END_WHILE
enumerator.Dispose();
END_METHOD

PROPERTY PUBLIC Address : PVOID
GET
Address := ADR(activeData);
END_GET
END_PROPERTY

PROPERTY PUBLIC BaseDatatype : I_Datatype
GET
BaseDatatype := baseType;
END_GET
END_PROPERTY

METHOD PUBLIC ClearReference
VAR_INPUT
END_VAR
activeData REF= localData;
SetElementReference();
END_METHOD

PROPERTY PUBLIC Size : UDINT
GET
Size := SIZEOF(activeData);
END_GET
END_PROPERTY

METHOD PUBLIC TryGetElementAsDatatypeByIndex : BOOL
VAR_INPUT
	Index : DINT;
	Destination : REFERENCE TO I_Datatype;
END_VAR
IF Index < lbound OR Index > ubound THEN
	RETURN;
END_IF

Destination := elements[Index];
TryGetElementAsDatatypeByIndex := TRUE;
END_METHOD

METHOD PUBLIC TryGetLowerBound : BOOL
VAR_INPUT
	Dimention : UDINT;
	Destination : REFERENCE TO DINT;
END_VAR
IF Dimention = 1 THEN
	Destination := lBound;
	TryGetLowerBound := TRUE;
END_IF
END_METHOD

METHOD PUBLIC TryGetUpperBound : BOOL
VAR_INPUT
	Dimention : UDINT;
	Destination : REFERENCE TO DINT;
END_VAR
IF Dimention = 1 THEN
	Destination := uBound;
	TryGetUpperBound := TRUE;
END_IF
END_METHOD

METHOD PUBLIC Clone : I_Datatype
VAR
    pClone : POINTER TO _Array0to3OfINT;
END_VAR
pClone := __NEW(_Array0to3OfINT());
pClone^.Value := Value;
Clone := pClone^;
END_METHOD

METHOD PUBLIC MakeReferenceTo
VAR_INPUT
	ReferenceTarget : REFERENCE TO ARRAY [lBound..uBound] OF INT;
END_VAR
activeData REF= ReferenceTarget;
SetElementReference();
END_METHOD

METHOD TryMakeReferenceTo : BOOL
VAR_INPUT
	Target : I_Datatype;
END_VAR
VAR
	targetAsArray : I_ArrayDatatype;
	pTargetData : POINTER TO ARRAY [lBound..uBound] OF INT;
END_VAR
IF NOT Target.TryResolveAsArrayDatatype(targetAsArray) THEN
	RETURN;
END_IF

IF NOT (targetAsArray.Identifier = Identifier) THEN
	RETURN;
END_IF

pTargetData := Target.Address;
activeData REF= pTargetData^;
SetElementReference();
TryMakeReferenceTo := TRUE;
END_METHOD

PROPERTY PUBLIC Value : REFERENCE TO ARRAY [lBound..uBound] OF INT;
GET
Value ref= activeData;
END_GET
END_PROPERTY

END_FUNCTION_BLOCK

// Datatypes/Aliases/_TcVnVector4_LREAL
{attribute 'linkalways'} 
{attribute 'no_explicit_call' := 'This FB is a CLASS and must be accessed using methods or properties'}
{attribute 'enable_dynamic_creation'}
FUNCTION_BLOCK _TcVnVector4_LREAL EXTENDS AliasDatatypeBase
VAR
	localData : TcVnVector4_LREAL;
	activeData : REFERENCE TO TcVnVector4_LREAL REF= localData;
	aliasBaseDatatype : _Array0to3OfLREAL;
END_VAR

METHOD PROTECTED SetBaseDatatypeReference
VAR_INPUT
END_VAR
aliasBaseDatatype.MakeReferenceTo(activeData);
END_METHOD

PROPERTY PUBLIC Address : PVOID
GET
Address := ADR(activeData);
END_GET
END_PROPERTY

METHOD PUBLIC ClearReference
VAR_INPUT
END_VAR
activeData REF= localData;
SetBaseDatatypeReference();
END_METHOD

PROPERTY PUBLIC Size : UDINT
GET
Size := SIZEOF(activeData);
END_GET
END_PROPERTY

METHOD FB_init : BOOL
VAR_INPUT
	bInitRetains : BOOL; // if TRUE, the retain variables are initialized (warm start / cold start)
	bInCopyCode : BOOL;  // if TRUE, the instance afterwards gets moved into the copy code (online change)
	//InitialValue : <type>; // if possible, not all values can be initialized
END_VAR
//localData := InitialValue; // if possible, not all values can be initialized
SetBaseDatatypeReference();
AddBaseDatatype(aliasBaseDatatype);
END_METHOD

METHOD PUBLIC Clone : I_Datatype
VAR
    pClone : POINTER TO _TcVnVector4_LREAL;
END_VAR
pClone := __NEW(_TcVnVector4_LREAL);
Clone := pClone^;
END_METHOD

PROPERTY PUBLIC Identifier : T_MAXSTRING
GET
Identifier := 'TcVnVector4_LREAL';
END_GET
END_PROPERTY

METHOD PUBLIC MakeReferenceTo
VAR_INPUT
	ReferenceTarget : REFERENCE TO TcVnVector4_LREAL;
END_VAR
activeData REF= ReferenceTarget;
SetBaseDatatypeReference();
END_METHOD

METHOD TryMakeReferenceTo : BOOL
VAR_INPUT
	Target : I_Datatype;
END_VAR
VAR
	targetAsAlias : I_AliasDatatype;
	pTargetData : POINTER TO TcVnVector4_LREAL;
END_VAR
IF NOT Target.TryResolveAsAliasDatatype(targetAsAlias) THEN
	RETURN;
END_IF

IF targetAsAlias.Identifier <> Identifier THEN
	RETURN;
END_IF

pTargetData := Target.Address;
activeData REF= pTargetData^;
SetBaseDatatypeReference();
TryMakeReferenceTo := TRUE;
END_METHOD

PROPERTY PUBLIC Value : REFERENCE TO TcVnVector4_LREAL
GET
Value REF= activeData;
END_GET
END_PROPERTY

END_FUNCTION_BLOCK

// Datatypes/Aliases/_TcVnVector4_SINT
{attribute 'linkalways'} 
{attribute 'no_explicit_call' := 'This FB is a CLASS and must be accessed using methods or properties'}
{attribute 'enable_dynamic_creation'}
FUNCTION_BLOCK _TcVnVector4_SINT EXTENDS AliasDatatypeBase
VAR
	localData : TcVnVector4_SINT;
	activeData : REFERENCE TO TcVnVector4_SINT REF= localData;
	aliasBaseDatatype : _Array0to3OfSINT;
END_VAR

METHOD PROTECTED SetBaseDatatypeReference
VAR_INPUT
END_VAR
aliasBaseDatatype.MakeReferenceTo(activeData);
END_METHOD

PROPERTY PUBLIC Address : PVOID
GET
Address := ADR(activeData);
END_GET
END_PROPERTY

METHOD PUBLIC ClearReference
VAR_INPUT
END_VAR
activeData REF= localData;
SetBaseDatatypeReference();
END_METHOD

PROPERTY PUBLIC Size : UDINT
GET
Size := SIZEOF(activeData);
END_GET
END_PROPERTY

METHOD FB_init : BOOL
VAR_INPUT
	bInitRetains : BOOL; // if TRUE, the retain variables are initialized (warm start / cold start)
	bInCopyCode : BOOL;  // if TRUE, the instance afterwards gets moved into the copy code (online change)
	//InitialValue : <type>; // if possible, not all values can be initialized
END_VAR
//localData := InitialValue; // if possible, not all values can be initialized
SetBaseDatatypeReference();
AddBaseDatatype(aliasBaseDatatype);
END_METHOD

METHOD PUBLIC Clone : I_Datatype
VAR
    pClone : POINTER TO _TcVnVector4_SINT;
END_VAR
pClone := __NEW(_TcVnVector4_SINT);
Clone := pClone^;
END_METHOD

PROPERTY PUBLIC Identifier : T_MAXSTRING
GET
Identifier := 'TcVnVector4_SINT';
END_GET
END_PROPERTY

METHOD PUBLIC MakeReferenceTo
VAR_INPUT
	ReferenceTarget : REFERENCE TO TcVnVector4_SINT;
END_VAR
activeData REF= ReferenceTarget;
SetBaseDatatypeReference();
END_METHOD

METHOD TryMakeReferenceTo : BOOL
VAR_INPUT
	Target : I_Datatype;
END_VAR
VAR
	targetAsAlias : I_AliasDatatype;
	pTargetData : POINTER TO TcVnVector4_SINT;
END_VAR
IF NOT Target.TryResolveAsAliasDatatype(targetAsAlias) THEN
	RETURN;
END_IF

IF targetAsAlias.Identifier <> Identifier THEN
	RETURN;
END_IF

pTargetData := Target.Address;
activeData REF= pTargetData^;
SetBaseDatatypeReference();
TryMakeReferenceTo := TRUE;
END_METHOD

PROPERTY PUBLIC Value : REFERENCE TO TcVnVector4_SINT
GET
Value REF= activeData;
END_GET
END_PROPERTY

END_FUNCTION_BLOCK

// Datatypes/Arrays/_Array0to3OfSINT
{attribute 'linkalways'} 
{attribute 'no_explicit_call' := 'This FB is a CLASS and must be accessed using methods or properties'}
{attribute 'enable_dynamic_creation'}
FUNCTION_BLOCK _Array0to3OfSINT EXTENDS ArrayDatatypeBase_1D
VAR CONSTANT
	lBound : DINT := 0;
	uBound : DINT := 3;
END_VAR
VAR
	localData : ARRAY [lBound..uBound] OF SINT;
	activeData : REFERENCE TO ARRAY [lBound..uBound] OF SINT REF= localData;
	elements : ARRAY [lBound..uBound] OF _SINT(0);
	baseType : _SINT(0);
END_VAR

METHOD FB_init : BOOL
VAR_INPUT
	bInitRetains : BOOL; // if TRUE, the retain variables are initialized (warm start / cold start)
	bInCopyCode : BOOL;  // if TRUE, the instance afterwards gets moved into the copy code (online change)
END_VAR
SetElementReference();
END_METHOD

METHOD PROTECTED OnSerializeArrayValues
VAR_INPUT
	Serializer : I_Serializer;
END_VAR
VAR
	i : DINT;
END_VAR
FOR i := lBound TO uBound DO
	elements[i].SerializeWith(Serializer);
END_FOR
END_METHOD

METHOD PROTECTED SetElementReference
VAR_INPUT
END_VAR
VAR
	i : DINT;
END_VAR
FOR i := lBound TO uBound DO
	elements[i].MakeReferenceTo(activeData[i]);
END_FOR
END_METHOD

METHOD PROTECTED TryDeserializeArrayValues : BOOL
VAR_INPUT
	Deserializer : I_Deserializer;
	Feedback : I_DeserializerFeedback;
END_VAR
VAR
	enumerator : I_DeserializerArrayForwardEnumerator;
	i : DINT;
END_VAR
enumerator := Deserializer.GetArrayEnumerator();
i := lBound;

WHILE enumerator.MoveNext() AND i <= uBound DO
	
	IF NOT elements[i].TryDeserializeFrom(enumerator.Current, Feedback) THEN
		EXIT;
	END_IF
	i := i + 1;

END_WHILE
enumerator.Dispose();
END_METHOD

PROPERTY PUBLIC Address : PVOID
GET
Address := ADR(activeData);
END_GET
END_PROPERTY

PROPERTY PUBLIC BaseDatatype : I_Datatype
GET
BaseDatatype := baseType;
END_GET
END_PROPERTY

METHOD PUBLIC ClearReference
VAR_INPUT
END_VAR
activeData REF= localData;
SetElementReference();
END_METHOD

PROPERTY PUBLIC Size : UDINT
GET
Size := SIZEOF(activeData);
END_GET
END_PROPERTY

METHOD PUBLIC TryGetElementAsDatatypeByIndex : BOOL
VAR_INPUT
	Index : DINT;
	Destination : REFERENCE TO I_Datatype;
END_VAR
IF Index < lbound OR Index > ubound THEN
	RETURN;
END_IF

Destination := elements[Index];
TryGetElementAsDatatypeByIndex := TRUE;
END_METHOD

METHOD PUBLIC TryGetLowerBound : BOOL
VAR_INPUT
	Dimention : UDINT;
	Destination : REFERENCE TO DINT;
END_VAR
IF Dimention = 1 THEN
	Destination := lBound;
	TryGetLowerBound := TRUE;
END_IF
END_METHOD

METHOD PUBLIC TryGetUpperBound : BOOL
VAR_INPUT
	Dimention : UDINT;
	Destination : REFERENCE TO DINT;
END_VAR
IF Dimention = 1 THEN
	Destination := uBound;
	TryGetUpperBound := TRUE;
END_IF
END_METHOD

METHOD PUBLIC Clone : I_Datatype
VAR
    pClone : POINTER TO _Array0to3OfSINT;
END_VAR
pClone := __NEW(_Array0to3OfSINT());
pClone^.Value := Value;
Clone := pClone^;
END_METHOD

METHOD PUBLIC MakeReferenceTo
VAR_INPUT
	ReferenceTarget : REFERENCE TO ARRAY [lBound..uBound] OF SINT;
END_VAR
activeData REF= ReferenceTarget;
SetElementReference();
END_METHOD

METHOD TryMakeReferenceTo : BOOL
VAR_INPUT
	Target : I_Datatype;
END_VAR
VAR
	targetAsArray : I_ArrayDatatype;
	pTargetData : POINTER TO ARRAY [lBound..uBound] OF SINT;
END_VAR
IF NOT Target.TryResolveAsArrayDatatype(targetAsArray) THEN
	RETURN;
END_IF

IF NOT (targetAsArray.Identifier = Identifier) THEN
	RETURN;
END_IF

pTargetData := Target.Address;
activeData REF= pTargetData^;
SetElementReference();
TryMakeReferenceTo := TRUE;
END_METHOD

PROPERTY PUBLIC Value : REFERENCE TO ARRAY [lBound..uBound] OF SINT;
GET
Value ref= activeData;
END_GET
END_PROPERTY

END_FUNCTION_BLOCK

// Datatypes/Aliases/_TcVnVector4_UINT
{attribute 'linkalways'} 
{attribute 'no_explicit_call' := 'This FB is a CLASS and must be accessed using methods or properties'}
{attribute 'enable_dynamic_creation'}
FUNCTION_BLOCK _TcVnVector4_UINT EXTENDS AliasDatatypeBase
VAR
	localData : TcVnVector4_UINT;
	activeData : REFERENCE TO TcVnVector4_UINT REF= localData;
	aliasBaseDatatype : _Array0to3OfUINT;
END_VAR

METHOD PROTECTED SetBaseDatatypeReference
VAR_INPUT
END_VAR
aliasBaseDatatype.MakeReferenceTo(activeData);
END_METHOD

PROPERTY PUBLIC Address : PVOID
GET
Address := ADR(activeData);
END_GET
END_PROPERTY

METHOD PUBLIC ClearReference
VAR_INPUT
END_VAR
activeData REF= localData;
SetBaseDatatypeReference();
END_METHOD

PROPERTY PUBLIC Size : UDINT
GET
Size := SIZEOF(activeData);
END_GET
END_PROPERTY

METHOD FB_init : BOOL
VAR_INPUT
	bInitRetains : BOOL; // if TRUE, the retain variables are initialized (warm start / cold start)
	bInCopyCode : BOOL;  // if TRUE, the instance afterwards gets moved into the copy code (online change)
	//InitialValue : <type>; // if possible, not all values can be initialized
END_VAR
//localData := InitialValue; // if possible, not all values can be initialized
SetBaseDatatypeReference();
AddBaseDatatype(aliasBaseDatatype);
END_METHOD

METHOD PUBLIC Clone : I_Datatype
VAR
    pClone : POINTER TO _TcVnVector4_UINT;
END_VAR
pClone := __NEW(_TcVnVector4_UINT);
Clone := pClone^;
END_METHOD

PROPERTY PUBLIC Identifier : T_MAXSTRING
GET
Identifier := 'TcVnVector4_UINT';
END_GET
END_PROPERTY

METHOD PUBLIC MakeReferenceTo
VAR_INPUT
	ReferenceTarget : REFERENCE TO TcVnVector4_UINT;
END_VAR
activeData REF= ReferenceTarget;
SetBaseDatatypeReference();
END_METHOD

METHOD TryMakeReferenceTo : BOOL
VAR_INPUT
	Target : I_Datatype;
END_VAR
VAR
	targetAsAlias : I_AliasDatatype;
	pTargetData : POINTER TO TcVnVector4_UINT;
END_VAR
IF NOT Target.TryResolveAsAliasDatatype(targetAsAlias) THEN
	RETURN;
END_IF

IF targetAsAlias.Identifier <> Identifier THEN
	RETURN;
END_IF

pTargetData := Target.Address;
activeData REF= pTargetData^;
SetBaseDatatypeReference();
TryMakeReferenceTo := TRUE;
END_METHOD

PROPERTY PUBLIC Value : REFERENCE TO TcVnVector4_UINT
GET
Value REF= activeData;
END_GET
END_PROPERTY

END_FUNCTION_BLOCK

// Datatypes/Arrays/_Array0to3OfUINT
{attribute 'linkalways'} 
{attribute 'no_explicit_call' := 'This FB is a CLASS and must be accessed using methods or properties'}
{attribute 'enable_dynamic_creation'}
FUNCTION_BLOCK _Array0to3OfUINT EXTENDS ArrayDatatypeBase_1D
VAR CONSTANT
	lBound : DINT := 0;
	uBound : DINT := 3;
END_VAR
VAR
	localData : ARRAY [lBound..uBound] OF UINT;
	activeData : REFERENCE TO ARRAY [lBound..uBound] OF UINT REF= localData;
	elements : ARRAY [lBound..uBound] OF _UINT(0);
	baseType : _UINT(0);
END_VAR

METHOD FB_init : BOOL
VAR_INPUT
	bInitRetains : BOOL; // if TRUE, the retain variables are initialized (warm start / cold start)
	bInCopyCode : BOOL;  // if TRUE, the instance afterwards gets moved into the copy code (online change)
END_VAR
SetElementReference();
END_METHOD

METHOD PROTECTED OnSerializeArrayValues
VAR_INPUT
	Serializer : I_Serializer;
END_VAR
VAR
	i : DINT;
END_VAR
FOR i := lBound TO uBound DO
	elements[i].SerializeWith(Serializer);
END_FOR
END_METHOD

METHOD PROTECTED SetElementReference
VAR_INPUT
END_VAR
VAR
	i : DINT;
END_VAR
FOR i := lBound TO uBound DO
	elements[i].MakeReferenceTo(activeData[i]);
END_FOR
END_METHOD

METHOD PROTECTED TryDeserializeArrayValues : BOOL
VAR_INPUT
	Deserializer : I_Deserializer;
	Feedback : I_DeserializerFeedback;
END_VAR
VAR
	enumerator : I_DeserializerArrayForwardEnumerator;
	i : DINT;
END_VAR
enumerator := Deserializer.GetArrayEnumerator();
i := lBound;

WHILE enumerator.MoveNext() AND i <= uBound DO
	
	IF NOT elements[i].TryDeserializeFrom(enumerator.Current, Feedback) THEN
		EXIT;
	END_IF
	i := i + 1;

END_WHILE
enumerator.Dispose();
END_METHOD

PROPERTY PUBLIC Address : PVOID
GET
Address := ADR(activeData);
END_GET
END_PROPERTY

PROPERTY PUBLIC BaseDatatype : I_Datatype
GET
BaseDatatype := baseType;
END_GET
END_PROPERTY

METHOD PUBLIC ClearReference
VAR_INPUT
END_VAR
activeData REF= localData;
SetElementReference();
END_METHOD

PROPERTY PUBLIC Size : UDINT
GET
Size := SIZEOF(activeData);
END_GET
END_PROPERTY

METHOD PUBLIC TryGetElementAsDatatypeByIndex : BOOL
VAR_INPUT
	Index : DINT;
	Destination : REFERENCE TO I_Datatype;
END_VAR
IF Index < lbound OR Index > ubound THEN
	RETURN;
END_IF

Destination := elements[Index];
TryGetElementAsDatatypeByIndex := TRUE;
END_METHOD

METHOD PUBLIC TryGetLowerBound : BOOL
VAR_INPUT
	Dimention : UDINT;
	Destination : REFERENCE TO DINT;
END_VAR
IF Dimention = 1 THEN
	Destination := lBound;
	TryGetLowerBound := TRUE;
END_IF
END_METHOD

METHOD PUBLIC TryGetUpperBound : BOOL
VAR_INPUT
	Dimention : UDINT;
	Destination : REFERENCE TO DINT;
END_VAR
IF Dimention = 1 THEN
	Destination := uBound;
	TryGetUpperBound := TRUE;
END_IF
END_METHOD

METHOD PUBLIC Clone : I_Datatype
VAR
    pClone : POINTER TO _Array0to3OfUINT;
END_VAR
pClone := __NEW(_Array0to3OfUINT());
pClone^.Value := Value;
Clone := pClone^;
END_METHOD

METHOD PUBLIC MakeReferenceTo
VAR_INPUT
	ReferenceTarget : REFERENCE TO ARRAY [lBound..uBound] OF UINT;
END_VAR
activeData REF= ReferenceTarget;
SetElementReference();
END_METHOD

METHOD TryMakeReferenceTo : BOOL
VAR_INPUT
	Target : I_Datatype;
END_VAR
VAR
	targetAsArray : I_ArrayDatatype;
	pTargetData : POINTER TO ARRAY [lBound..uBound] OF UINT;
END_VAR
IF NOT Target.TryResolveAsArrayDatatype(targetAsArray) THEN
	RETURN;
END_IF

IF NOT (targetAsArray.Identifier = Identifier) THEN
	RETURN;
END_IF

pTargetData := Target.Address;
activeData REF= pTargetData^;
SetElementReference();
TryMakeReferenceTo := TRUE;
END_METHOD

PROPERTY PUBLIC Value : REFERENCE TO ARRAY [lBound..uBound] OF UINT;
GET
Value ref= activeData;
END_GET
END_PROPERTY

END_FUNCTION_BLOCK

// Datatypes/Aliases/_TcVnVector4_USINT
{attribute 'linkalways'} 
{attribute 'no_explicit_call' := 'This FB is a CLASS and must be accessed using methods or properties'}
{attribute 'enable_dynamic_creation'}
FUNCTION_BLOCK _TcVnVector4_USINT EXTENDS AliasDatatypeBase
VAR
	localData : TcVnVector4_USINT;
	activeData : REFERENCE TO TcVnVector4_USINT REF= localData;
	aliasBaseDatatype : _Array0to3OfUSINT;
END_VAR

METHOD PROTECTED SetBaseDatatypeReference
VAR_INPUT
END_VAR
aliasBaseDatatype.MakeReferenceTo(activeData);
END_METHOD

PROPERTY PUBLIC Address : PVOID
GET
Address := ADR(activeData);
END_GET
END_PROPERTY

METHOD PUBLIC ClearReference
VAR_INPUT
END_VAR
activeData REF= localData;
SetBaseDatatypeReference();
END_METHOD

PROPERTY PUBLIC Size : UDINT
GET
Size := SIZEOF(activeData);
END_GET
END_PROPERTY

METHOD FB_init : BOOL
VAR_INPUT
	bInitRetains : BOOL; // if TRUE, the retain variables are initialized (warm start / cold start)
	bInCopyCode : BOOL;  // if TRUE, the instance afterwards gets moved into the copy code (online change)
	//InitialValue : <type>; // if possible, not all values can be initialized
END_VAR
//localData := InitialValue; // if possible, not all values can be initialized
SetBaseDatatypeReference();
AddBaseDatatype(aliasBaseDatatype);
END_METHOD

METHOD PUBLIC Clone : I_Datatype
VAR
    pClone : POINTER TO _TcVnVector4_USINT;
END_VAR
pClone := __NEW(_TcVnVector4_USINT);
Clone := pClone^;
END_METHOD

PROPERTY PUBLIC Identifier : T_MAXSTRING
GET
Identifier := 'TcVnVector4_USINT';
END_GET
END_PROPERTY

METHOD PUBLIC MakeReferenceTo
VAR_INPUT
	ReferenceTarget : REFERENCE TO TcVnVector4_USINT;
END_VAR
activeData REF= ReferenceTarget;
SetBaseDatatypeReference();
END_METHOD

METHOD TryMakeReferenceTo : BOOL
VAR_INPUT
	Target : I_Datatype;
END_VAR
VAR
	targetAsAlias : I_AliasDatatype;
	pTargetData : POINTER TO TcVnVector4_USINT;
END_VAR
IF NOT Target.TryResolveAsAliasDatatype(targetAsAlias) THEN
	RETURN;
END_IF

IF targetAsAlias.Identifier <> Identifier THEN
	RETURN;
END_IF

pTargetData := Target.Address;
activeData REF= pTargetData^;
SetBaseDatatypeReference();
TryMakeReferenceTo := TRUE;
END_METHOD

PROPERTY PUBLIC Value : REFERENCE TO TcVnVector4_USINT
GET
Value REF= activeData;
END_GET
END_PROPERTY

END_FUNCTION_BLOCK

// Datatypes/Arrays/_Array0to3OfUSINT
{attribute 'linkalways'} 
{attribute 'no_explicit_call' := 'This FB is a CLASS and must be accessed using methods or properties'}
{attribute 'enable_dynamic_creation'}
FUNCTION_BLOCK _Array0to3OfUSINT EXTENDS ArrayDatatypeBase_1D
VAR CONSTANT
	lBound : DINT := 0;
	uBound : DINT := 3;
END_VAR
VAR
	localData : ARRAY [lBound..uBound] OF USINT;
	activeData : REFERENCE TO ARRAY [lBound..uBound] OF USINT REF= localData;
	elements : ARRAY [lBound..uBound] OF _USINT(0);
	baseType : _USINT(0);
END_VAR

METHOD FB_init : BOOL
VAR_INPUT
	bInitRetains : BOOL; // if TRUE, the retain variables are initialized (warm start / cold start)
	bInCopyCode : BOOL;  // if TRUE, the instance afterwards gets moved into the copy code (online change)
END_VAR
SetElementReference();
END_METHOD

METHOD PROTECTED OnSerializeArrayValues
VAR_INPUT
	Serializer : I_Serializer;
END_VAR
VAR
	i : DINT;
END_VAR
FOR i := lBound TO uBound DO
	elements[i].SerializeWith(Serializer);
END_FOR
END_METHOD

METHOD PROTECTED SetElementReference
VAR_INPUT
END_VAR
VAR
	i : DINT;
END_VAR
FOR i := lBound TO uBound DO
	elements[i].MakeReferenceTo(activeData[i]);
END_FOR
END_METHOD

METHOD PROTECTED TryDeserializeArrayValues : BOOL
VAR_INPUT
	Deserializer : I_Deserializer;
	Feedback : I_DeserializerFeedback;
END_VAR
VAR
	enumerator : I_DeserializerArrayForwardEnumerator;
	i : DINT;
END_VAR
enumerator := Deserializer.GetArrayEnumerator();
i := lBound;

WHILE enumerator.MoveNext() AND i <= uBound DO
	
	IF NOT elements[i].TryDeserializeFrom(enumerator.Current, Feedback) THEN
		EXIT;
	END_IF
	i := i + 1;

END_WHILE
enumerator.Dispose();
END_METHOD

PROPERTY PUBLIC Address : PVOID
GET
Address := ADR(activeData);
END_GET
END_PROPERTY

PROPERTY PUBLIC BaseDatatype : I_Datatype
GET
BaseDatatype := baseType;
END_GET
END_PROPERTY

METHOD PUBLIC ClearReference
VAR_INPUT
END_VAR
activeData REF= localData;
SetElementReference();
END_METHOD

PROPERTY PUBLIC Size : UDINT
GET
Size := SIZEOF(activeData);
END_GET
END_PROPERTY

METHOD PUBLIC TryGetElementAsDatatypeByIndex : BOOL
VAR_INPUT
	Index : DINT;
	Destination : REFERENCE TO I_Datatype;
END_VAR
IF Index < lbound OR Index > ubound THEN
	RETURN;
END_IF

Destination := elements[Index];
TryGetElementAsDatatypeByIndex := TRUE;
END_METHOD

METHOD PUBLIC TryGetLowerBound : BOOL
VAR_INPUT
	Dimention : UDINT;
	Destination : REFERENCE TO DINT;
END_VAR
IF Dimention = 1 THEN
	Destination := lBound;
	TryGetLowerBound := TRUE;
END_IF
END_METHOD

METHOD PUBLIC TryGetUpperBound : BOOL
VAR_INPUT
	Dimention : UDINT;
	Destination : REFERENCE TO DINT;
END_VAR
IF Dimention = 1 THEN
	Destination := uBound;
	TryGetUpperBound := TRUE;
END_IF
END_METHOD

METHOD PUBLIC Clone : I_Datatype
VAR
    pClone : POINTER TO _Array0to3OfUSINT;
END_VAR
pClone := __NEW(_Array0to3OfUSINT());
pClone^.Value := Value;
Clone := pClone^;
END_METHOD

METHOD PUBLIC MakeReferenceTo
VAR_INPUT
	ReferenceTarget : REFERENCE TO ARRAY [lBound..uBound] OF USINT;
END_VAR
activeData REF= ReferenceTarget;
SetElementReference();
END_METHOD

METHOD TryMakeReferenceTo : BOOL
VAR_INPUT
	Target : I_Datatype;
END_VAR
VAR
	targetAsArray : I_ArrayDatatype;
	pTargetData : POINTER TO ARRAY [lBound..uBound] OF USINT;
END_VAR
IF NOT Target.TryResolveAsArrayDatatype(targetAsArray) THEN
	RETURN;
END_IF

IF NOT (targetAsArray.Identifier = Identifier) THEN
	RETURN;
END_IF

pTargetData := Target.Address;
activeData REF= pTargetData^;
SetElementReference();
TryMakeReferenceTo := TRUE;
END_METHOD

PROPERTY PUBLIC Value : REFERENCE TO ARRAY [lBound..uBound] OF USINT;
GET
Value ref= activeData;
END_GET
END_PROPERTY

END_FUNCTION_BLOCK

// Datatypes/Arrays/_Array0to1_0to2OfLREAL
{attribute 'linkalways'} 
{attribute 'no_explicit_call' := 'This FB is a CLASS and must be accessed using methods or properties'}
{attribute 'enable_dynamic_creation'}
FUNCTION_BLOCK _Array0to1_0to2OfLREAL EXTENDS ArrayDatatypeBase_2D
VAR CONSTANT
	lBoundD1 : DINT := 0;
	uBoundD1 : DINT := 1;
	lBoundD2 : DINT := 0;
	uBoundD2 : DINT := 2;
END_VAR
VAR
	localData : ARRAY [lBoundD1..uBoundD1,lBoundD2..uBoundD2] OF LREAL;
	activeData : REFERENCE TO ARRAY [lBoundD1..uBoundD1,lBoundD2..uBoundD2] OF LREAL REF= localData;
	elements : ARRAY [lBoundD1..uBoundD1,lBoundD2..uBoundD2] OF _LREAL(0);
	baseType : _LREAL(0);
END_VAR

METHOD FB_init : BOOL
VAR_INPUT
	bInitRetains : BOOL; // if TRUE, the retain variables are initialized (warm start / cold start)
	bInCopyCode : BOOL;  // if TRUE, the instance afterwards gets moved into the copy code (online change)
END_VAR
SetElementReference();
END_METHOD

METHOD PROTECTED OnSerializeArrayValues
VAR_INPUT
	Serializer : I_Serializer;
END_VAR
VAR
	i, j : DINT;
END_VAR
FOR i := lBoundD1 TO uBoundD1 DO
	Serializer.StartArray();
	FOR j := lBoundD2 TO uBoundD2 DO
		elements[i, j].SerializeWith(Serializer);
	END_FOR
	Serializer.EndArray();
END_FOR
END_METHOD

METHOD PROTECTED SetElementReference
VAR_INPUT
END_VAR
VAR
	i, j : DINT;
END_VAR
FOR i := lBoundD1 TO uBoundD1 DO
	FOR j := lBoundD2 TO uBoundD2 DO
		elements[i, j].MakeReferenceTo(activeData[i, j]);
	END_FOR
END_FOR
END_METHOD

METHOD PROTECTED TryDeserializeArrayValues : BOOL
VAR_INPUT
	Deserializer : I_Deserializer;
	Feedback : I_DeserializerFeedback;
END_VAR
VAR
	enumeratorD1 : I_DeserializerArrayForwardEnumerator;
	enumeratorD2 : I_DeserializerArrayForwardEnumerator;
	i, j : DINT;
END_VAR
enumeratorD1 := Deserializer.GetArrayEnumerator();
i := lBoundD1;

WHILE enumeratorD1.MoveNext() AND i <= uBoundD1 DO
	
	enumeratorD2 := enumeratorD1.Current.GetArrayEnumerator();
	j := lBoundD2;
	
	WHILE enumeratorD2.MoveNext() AND j <= uBoundD2 DO
	
		IF NOT elements[i, j].TryDeserializeFrom(enumeratorD2.Current, Feedback) THEN
			EXIT;
		END_IF
		
		j := j + 1;
	
	END_WHILE
	enumeratorD2.Dispose();

	i := i + 1;

END_WHILE
enumeratorD1.Dispose();
END_METHOD

PROPERTY PUBLIC Address : PVOID
GET
Address := ADR(activeData);
END_GET
END_PROPERTY

PROPERTY PUBLIC BaseDatatype : I_Datatype
GET
BaseDatatype := baseType;
END_GET
END_PROPERTY

METHOD PUBLIC ClearReference
VAR_INPUT
END_VAR
activeData REF= localData;
SetElementReference();
END_METHOD

PROPERTY PUBLIC Size : UDINT
GET
Size := SIZEOF(activeData);
END_GET
END_PROPERTY

METHOD PUBLIC TryGetElementAsDatatypeByIndex : BOOL
VAR_INPUT
	Index1 : DINT;
	Index2 : DINT;
	Destination : REFERENCE TO I_Datatype;
END_VAR
IF Index1 < lboundD1 OR Index1 > uboundD1 THEN
	RETURN;
END_IF

IF Index2 < lboundD2 OR Index2 > uboundD2 THEN
	RETURN;
END_IF

Destination := elements[Index1, Index2];
TryGetElementAsDatatypeByIndex := TRUE;
END_METHOD

METHOD PUBLIC TryGetLowerBound : BOOL
VAR_INPUT
	Dimention : UDINT;
	Destination : REFERENCE TO DINT;
END_VAR
CASE Dimention OF
	
	1:	Destination := lBoundD1;
		TryGetLowerBound := TRUE;
		RETURN;
	
	2:	Destination := lBoundD2;
		TryGetLowerBound := TRUE;
		RETURN;

END_CASE
END_METHOD

METHOD PUBLIC TryGetUpperBound : BOOL
VAR_INPUT
	Dimention : UDINT;
	Destination : REFERENCE TO DINT;
END_VAR
CASE Dimention OF
	
	1:	Destination := uBoundD1;
		TryGetUpperBound := TRUE;
		RETURN;
	
	2:	Destination := uBoundD2;
		TryGetUpperBound := TRUE;
		RETURN;

END_CASE
END_METHOD

METHOD PUBLIC Clone : I_Datatype
VAR
    pClone : POINTER TO _Array0to1_0to2OfLREAL;
END_VAR
pClone := __NEW(_Array0to1_0to2OfLREAL());
pClone^.Value := Value;
Clone := pClone^;
END_METHOD

METHOD PUBLIC MakeReferenceTo
VAR_INPUT
	ReferenceTarget : REFERENCE TO ARRAY [lBoundD1..uBoundD1,lBoundD2..uBoundD2] OF LREAL;
END_VAR
activeData REF= ReferenceTarget;
SetElementReference();
END_METHOD

METHOD TryMakeReferenceTo : BOOL
VAR_INPUT
	Target : I_Datatype;
END_VAR
VAR
	targetAsArray : I_ArrayDatatype;
	pTargetData : POINTER TO ARRAY [lBoundD1..uBoundD1,lBoundD2..uBoundD2] OF LREAL;
END_VAR
IF NOT Target.TryResolveAsArrayDatatype(targetAsArray) THEN
	RETURN;
END_IF

IF NOT (targetAsArray.Identifier = Identifier) THEN
	RETURN;
END_IF

pTargetData := Target.Address;
activeData REF= pTargetData^;
SetElementReference();
TryMakeReferenceTo := TRUE;
END_METHOD

PROPERTY PUBLIC Value : REFERENCE TO ARRAY [lBoundD1..uBoundD1,lBoundD2..uBoundD2] OF LREAL;
GET
Value ref= activeData;
END_GET
END_PROPERTY

END_FUNCTION_BLOCK

// Datatypes/Arrays/_Array0to2_0to2OfLREAL
{attribute 'linkalways'} 
{attribute 'no_explicit_call' := 'This FB is a CLASS and must be accessed using methods or properties'}
{attribute 'enable_dynamic_creation'}
FUNCTION_BLOCK _Array0to2_0to2OfLREAL EXTENDS ArrayDatatypeBase_2D
VAR CONSTANT
	lBoundD1 : DINT := 0;
	uBoundD1 : DINT := 2;
	lBoundD2 : DINT := 0;
	uBoundD2 : DINT := 2;
END_VAR
VAR
	localData : ARRAY [lBoundD1..uBoundD1,lBoundD2..uBoundD2] OF LREAL;
	activeData : REFERENCE TO ARRAY [lBoundD1..uBoundD1,lBoundD2..uBoundD2] OF LREAL REF= localData;
	elements : ARRAY [lBoundD1..uBoundD1,lBoundD2..uBoundD2] OF _LREAL(0);
	baseType : _LREAL(0);
END_VAR

METHOD FB_init : BOOL
VAR_INPUT
	bInitRetains : BOOL; // if TRUE, the retain variables are initialized (warm start / cold start)
	bInCopyCode : BOOL;  // if TRUE, the instance afterwards gets moved into the copy code (online change)
END_VAR
SetElementReference();
END_METHOD

METHOD PROTECTED OnSerializeArrayValues
VAR_INPUT
	Serializer : I_Serializer;
END_VAR
VAR
	i, j : DINT;
END_VAR
FOR i := lBoundD1 TO uBoundD1 DO
	Serializer.StartArray();
	FOR j := lBoundD2 TO uBoundD2 DO
		elements[i, j].SerializeWith(Serializer);
	END_FOR
	Serializer.EndArray();
END_FOR
END_METHOD

METHOD PROTECTED SetElementReference
VAR_INPUT
END_VAR
VAR
	i, j : DINT;
END_VAR
FOR i := lBoundD1 TO uBoundD1 DO
	FOR j := lBoundD2 TO uBoundD2 DO
		elements[i, j].MakeReferenceTo(activeData[i, j]);
	END_FOR
END_FOR
END_METHOD

METHOD PROTECTED TryDeserializeArrayValues : BOOL
VAR_INPUT
	Deserializer : I_Deserializer;
	Feedback : I_DeserializerFeedback;
END_VAR
VAR
	enumeratorD1 : I_DeserializerArrayForwardEnumerator;
	enumeratorD2 : I_DeserializerArrayForwardEnumerator;
	i, j : DINT;
END_VAR
enumeratorD1 := Deserializer.GetArrayEnumerator();
i := lBoundD1;

WHILE enumeratorD1.MoveNext() AND i <= uBoundD1 DO
	
	enumeratorD2 := enumeratorD1.Current.GetArrayEnumerator();
	j := lBoundD2;
	
	WHILE enumeratorD2.MoveNext() AND j <= uBoundD2 DO
	
		IF NOT elements[i, j].TryDeserializeFrom(enumeratorD2.Current, Feedback) THEN
			EXIT;
		END_IF
		
		j := j + 1;
	
	END_WHILE
	enumeratorD2.Dispose();

	i := i + 1;

END_WHILE
enumeratorD1.Dispose();
END_METHOD

PROPERTY PUBLIC Address : PVOID
GET
Address := ADR(activeData);
END_GET
END_PROPERTY

PROPERTY PUBLIC BaseDatatype : I_Datatype
GET
BaseDatatype := baseType;
END_GET
END_PROPERTY

METHOD PUBLIC ClearReference
VAR_INPUT
END_VAR
activeData REF= localData;
SetElementReference();
END_METHOD

PROPERTY PUBLIC Size : UDINT
GET
Size := SIZEOF(activeData);
END_GET
END_PROPERTY

METHOD PUBLIC TryGetElementAsDatatypeByIndex : BOOL
VAR_INPUT
	Index1 : DINT;
	Index2 : DINT;
	Destination : REFERENCE TO I_Datatype;
END_VAR
IF Index1 < lboundD1 OR Index1 > uboundD1 THEN
	RETURN;
END_IF

IF Index2 < lboundD2 OR Index2 > uboundD2 THEN
	RETURN;
END_IF

Destination := elements[Index1, Index2];
TryGetElementAsDatatypeByIndex := TRUE;
END_METHOD

METHOD PUBLIC TryGetLowerBound : BOOL
VAR_INPUT
	Dimention : UDINT;
	Destination : REFERENCE TO DINT;
END_VAR
CASE Dimention OF
	
	1:	Destination := lBoundD1;
		TryGetLowerBound := TRUE;
		RETURN;
	
	2:	Destination := lBoundD2;
		TryGetLowerBound := TRUE;
		RETURN;

END_CASE
END_METHOD

METHOD PUBLIC TryGetUpperBound : BOOL
VAR_INPUT
	Dimention : UDINT;
	Destination : REFERENCE TO DINT;
END_VAR
CASE Dimention OF
	
	1:	Destination := uBoundD1;
		TryGetUpperBound := TRUE;
		RETURN;
	
	2:	Destination := uBoundD2;
		TryGetUpperBound := TRUE;
		RETURN;

END_CASE
END_METHOD

METHOD PUBLIC Clone : I_Datatype
VAR
    pClone : POINTER TO _Array0to2_0to2OfLREAL;
END_VAR
pClone := __NEW(_Array0to2_0to2OfLREAL());
pClone^.Value := Value;
Clone := pClone^;
END_METHOD

METHOD PUBLIC MakeReferenceTo
VAR_INPUT
	ReferenceTarget : REFERENCE TO ARRAY [lBoundD1..uBoundD1,lBoundD2..uBoundD2] OF LREAL;
END_VAR
activeData REF= ReferenceTarget;
SetElementReference();
END_METHOD

METHOD TryMakeReferenceTo : BOOL
VAR_INPUT
	Target : I_Datatype;
END_VAR
VAR
	targetAsArray : I_ArrayDatatype;
	pTargetData : POINTER TO ARRAY [lBoundD1..uBoundD1,lBoundD2..uBoundD2] OF LREAL;
END_VAR
IF NOT Target.TryResolveAsArrayDatatype(targetAsArray) THEN
	RETURN;
END_IF

IF NOT (targetAsArray.Identifier = Identifier) THEN
	RETURN;
END_IF

pTargetData := Target.Address;
activeData REF= pTargetData^;
SetElementReference();
TryMakeReferenceTo := TRUE;
END_METHOD

PROPERTY PUBLIC Value : REFERENCE TO ARRAY [lBoundD1..uBoundD1,lBoundD2..uBoundD2] OF LREAL;
GET
Value ref= activeData;
END_GET
END_PROPERTY

END_FUNCTION_BLOCK

// Datatypes/Arrays/_Array0to32OfUDINT
{attribute 'linkalways'} 
{attribute 'no_explicit_call' := 'This FB is a CLASS and must be accessed using methods or properties'}
{attribute 'enable_dynamic_creation'}
FUNCTION_BLOCK _Array0to32OfUDINT EXTENDS ArrayDatatypeBase_1D
VAR CONSTANT
	lBound : DINT := 0;
	uBound : DINT := 32;
END_VAR
VAR
	localData : ARRAY [lBound..uBound] OF UDINT;
	activeData : REFERENCE TO ARRAY [lBound..uBound] OF UDINT REF= localData;
	elements : ARRAY [lBound..uBound] OF _UDINT(0);
	baseType : _UDINT(0);
END_VAR

METHOD FB_init : BOOL
VAR_INPUT
	bInitRetains : BOOL; // if TRUE, the retain variables are initialized (warm start / cold start)
	bInCopyCode : BOOL;  // if TRUE, the instance afterwards gets moved into the copy code (online change)
END_VAR
SetElementReference();
END_METHOD

METHOD PROTECTED OnSerializeArrayValues
VAR_INPUT
	Serializer : I_Serializer;
END_VAR
VAR
	i : DINT;
END_VAR
FOR i := lBound TO uBound DO
	elements[i].SerializeWith(Serializer);
END_FOR
END_METHOD

METHOD PROTECTED SetElementReference
VAR_INPUT
END_VAR
VAR
	i : DINT;
END_VAR
FOR i := lBound TO uBound DO
	elements[i].MakeReferenceTo(activeData[i]);
END_FOR
END_METHOD

METHOD PROTECTED TryDeserializeArrayValues : BOOL
VAR_INPUT
	Deserializer : I_Deserializer;
	Feedback : I_DeserializerFeedback;
END_VAR
VAR
	enumerator : I_DeserializerArrayForwardEnumerator;
	i : DINT;
END_VAR
enumerator := Deserializer.GetArrayEnumerator();
i := lBound;

WHILE enumerator.MoveNext() AND i <= uBound DO
	
	IF NOT elements[i].TryDeserializeFrom(enumerator.Current, Feedback) THEN
		EXIT;
	END_IF
	i := i + 1;

END_WHILE
enumerator.Dispose();
END_METHOD

PROPERTY PUBLIC Address : PVOID
GET
Address := ADR(activeData);
END_GET
END_PROPERTY

PROPERTY PUBLIC BaseDatatype : I_Datatype
GET
BaseDatatype := baseType;
END_GET
END_PROPERTY

METHOD PUBLIC ClearReference
VAR_INPUT
END_VAR
activeData REF= localData;
SetElementReference();
END_METHOD

PROPERTY PUBLIC Size : UDINT
GET
Size := SIZEOF(activeData);
END_GET
END_PROPERTY

METHOD PUBLIC TryGetElementAsDatatypeByIndex : BOOL
VAR_INPUT
	Index : DINT;
	Destination : REFERENCE TO I_Datatype;
END_VAR
IF Index < lbound OR Index > ubound THEN
	RETURN;
END_IF

Destination := elements[Index];
TryGetElementAsDatatypeByIndex := TRUE;
END_METHOD

METHOD PUBLIC TryGetLowerBound : BOOL
VAR_INPUT
	Dimention : UDINT;
	Destination : REFERENCE TO DINT;
END_VAR
IF Dimention = 1 THEN
	Destination := lBound;
	TryGetLowerBound := TRUE;
END_IF
END_METHOD

METHOD PUBLIC TryGetUpperBound : BOOL
VAR_INPUT
	Dimention : UDINT;
	Destination : REFERENCE TO DINT;
END_VAR
IF Dimention = 1 THEN
	Destination := uBound;
	TryGetUpperBound := TRUE;
END_IF
END_METHOD

METHOD PUBLIC Clone : I_Datatype
VAR
    pClone : POINTER TO _Array0to32OfUDINT;
END_VAR
pClone := __NEW(_Array0to32OfUDINT());
pClone^.Value := Value;
Clone := pClone^;
END_METHOD

METHOD PUBLIC MakeReferenceTo
VAR_INPUT
	ReferenceTarget : REFERENCE TO ARRAY [lBound..uBound] OF UDINT;
END_VAR
activeData REF= ReferenceTarget;
SetElementReference();
END_METHOD

METHOD TryMakeReferenceTo : BOOL
VAR_INPUT
	Target : I_Datatype;
END_VAR
VAR
	targetAsArray : I_ArrayDatatype;
	pTargetData : POINTER TO ARRAY [lBound..uBound] OF UDINT;
END_VAR
IF NOT Target.TryResolveAsArrayDatatype(targetAsArray) THEN
	RETURN;
END_IF

IF NOT (targetAsArray.Identifier = Identifier) THEN
	RETURN;
END_IF

pTargetData := Target.Address;
activeData REF= pTargetData^;
SetElementReference();
TryMakeReferenceTo := TRUE;
END_METHOD

PROPERTY PUBLIC Value : REFERENCE TO ARRAY [lBound..uBound] OF UDINT;
GET
Value ref= activeData;
END_GET
END_PROPERTY

END_FUNCTION_BLOCK

// Datatypes/Enums/_ETcVn2dCodeSearchStrategy
{attribute 'linkalways'} 
{attribute 'no_explicit_call' := 'This FB is a CLASS and must be accessed using methods or properties'}
{attribute 'enable_dynamic_creation'}
FUNCTION_BLOCK _ETcVn2dCodeSearchStrategy EXTENDS EnumDatatypeBase
VAR
	localData : ETcVn2dCodeSearchStrategy;
	activeData : REFERENCE TO ETcVn2dCodeSearchStrategy;
	enumBaseDatatype : _UDINT(localData);
END_VAR

METHOD PROTECTED SetBaseDatatypeReference
VAR_INPUT
END_VAR
enumBaseDatatype.MakeReferenceTo(activeData);
END_METHOD

PROPERTY PUBLIC Address : PVOID
GET
Address := ADR(activeData);
END_GET
END_PROPERTY

METHOD PUBLIC ClearReference
VAR_INPUT
END_VAR
activeData REF= localData;
SetBaseDatatypeReference();
END_METHOD

PROPERTY PUBLIC Size : UDINT
GET
Size := SIZEOF(activeData);
END_GET
END_PROPERTY

METHOD FB_init : BOOL
VAR_INPUT
	bInitRetains : BOOL; // if TRUE, the retain variables are initialized (warm start / cold start)
	bInCopyCode : BOOL;  // if TRUE, the instance afterwards gets moved into the copy code (online change)
	InitialValue : ETcVn2dCodeSearchStrategy;
END_VAR
localData := InitialValue;
AddBaseDatatype(enumBaseDatatype);
ClearReference();

AddLocalEnumeration('TCVN_CSS_DEFAULT', ETcVn2dCodeSearchStrategy.TCVN_CSS_DEFAULT);
AddLocalEnumeration('TCVN_CSS_FIRST_FLIPPED', ETcVn2dCodeSearchStrategy.TCVN_CSS_FIRST_FLIPPED);
AddLocalEnumeration('TCVN_CSS_FIRST_INVERTED', ETcVn2dCodeSearchStrategy.TCVN_CSS_FIRST_INVERTED);
AddLocalEnumeration('TCVN_CSS_FIRST_NOT_FLIPPED', ETcVn2dCodeSearchStrategy.TCVN_CSS_FIRST_NOT_FLIPPED);
AddLocalEnumeration('TCVN_CSS_FIRST_NOT_INVERTED', ETcVn2dCodeSearchStrategy.TCVN_CSS_FIRST_NOT_INVERTED);
AddLocalEnumeration('TCVN_CSS_ONLY_FLIPPED', ETcVn2dCodeSearchStrategy.TCVN_CSS_ONLY_FLIPPED);
AddLocalEnumeration('TCVN_CSS_ONLY_INVERTED', ETcVn2dCodeSearchStrategy.TCVN_CSS_ONLY_INVERTED);
AddLocalEnumeration('TCVN_CSS_ONLY_NOT_FLIPPED', ETcVn2dCodeSearchStrategy.TCVN_CSS_ONLY_NOT_FLIPPED);
AddLocalEnumeration('TCVN_CSS_ONLY_NOT_INVERTED', ETcVn2dCodeSearchStrategy.TCVN_CSS_ONLY_NOT_INVERTED);
END_METHOD

METHOD PRIVATE AddLocalEnumeration
VAR_INPUT
	Enumeration : T_MAXSTRING;
	Value : ETcVn2dCodeSearchStrategy;
END_VAR
AddEnumeration(Enumeration, Value);
END_METHOD

METHOD IsEnumeratorValueEqual : BOOL
VAR_INPUT
	Enumerator : I_KeyValueForwardEnumerator;
END_VAR
VAR
	storedValue : ETcVn2dCodeSearchStrategy;
END_VAR
IF NOT Enumerator.TryGet(storedValue) THEN
	RETURN;
END_IF

IsEnumeratorValueEqual := storedValue = activeData;
END_METHOD

METHOD PUBLIC Clone : I_Datatype
VAR
    pClone : POINTER TO _ETcVn2dCodeSearchStrategy;
END_VAR
pClone := __NEW(_ETcVn2dCodeSearchStrategy(InitialValue := Value));
Clone := pClone^;
END_METHOD

PROPERTY PUBLIC Identifier : T_MAXSTRING
GET
Identifier := 'ETcVn2dCodeSearchStrategy';
END_GET
END_PROPERTY

METHOD PUBLIC MakeReferenceTo
VAR_INPUT
	ReferenceTarget : REFERENCE TO ETcVn2dCodeSearchStrategy;
END_VAR
activeData REF= ReferenceTarget;
SetBaseDatatypeReference();
END_METHOD

METHOD TryMakeReferenceTo : BOOL
VAR_INPUT
	Target : I_Datatype;
END_VAR
VAR
	targetAsEnum : I_EnumDatatype;
	pTargetData : POINTER TO ETcVn2dCodeSearchStrategy;
END_VAR
IF NOT Target.TryResolveAsEnumDatatype(targetAsEnum) THEN
	RETURN;
END_IF

IF targetAsEnum.Identifier <> Identifier THEN
	RETURN;
END_IF

pTargetData := Target.Address;
activeData REF= pTargetData^;
SetBaseDatatypeReference();
TryMakeReferenceTo := TRUE;
END_METHOD

PROPERTY PUBLIC Value : ETcVn2dCodeSearchStrategy
GET
Value := activeData;
END_GET
SET
activeData := Value;
END_SET
END_PROPERTY

END_FUNCTION_BLOCK

// Datatypes/Enums/_ETcVnAdaptiveThresholdMethod
{attribute 'linkalways'} 
{attribute 'no_explicit_call' := 'This FB is a CLASS and must be accessed using methods or properties'}
{attribute 'enable_dynamic_creation'}
FUNCTION_BLOCK _ETcVnAdaptiveThresholdMethod EXTENDS EnumDatatypeBase
VAR
	localData : ETcVnAdaptiveThresholdMethod;
	activeData : REFERENCE TO ETcVnAdaptiveThresholdMethod;
	enumBaseDatatype : _DINT(localData);
END_VAR

METHOD PROTECTED SetBaseDatatypeReference
VAR_INPUT
END_VAR
enumBaseDatatype.MakeReferenceTo(activeData);
END_METHOD

PROPERTY PUBLIC Address : PVOID
GET
Address := ADR(activeData);
END_GET
END_PROPERTY

METHOD PUBLIC ClearReference
VAR_INPUT
END_VAR
activeData REF= localData;
SetBaseDatatypeReference();
END_METHOD

PROPERTY PUBLIC Size : UDINT
GET
Size := SIZEOF(activeData);
END_GET
END_PROPERTY

METHOD FB_init : BOOL
VAR_INPUT
	bInitRetains : BOOL; // if TRUE, the retain variables are initialized (warm start / cold start)
	bInCopyCode : BOOL;  // if TRUE, the instance afterwards gets moved into the copy code (online change)
	InitialValue : ETcVnAdaptiveThresholdMethod;
END_VAR
localData := InitialValue;
AddBaseDatatype(enumBaseDatatype);
ClearReference();

AddLocalEnumeration('TCVN_ATM_MEAN', ETcVnAdaptiveThresholdMethod.TCVN_ATM_MEAN);
AddLocalEnumeration('TCVN_ATM_GAUSSIAN', ETcVnAdaptiveThresholdMethod.TCVN_ATM_GAUSSIAN);
END_METHOD

METHOD PRIVATE AddLocalEnumeration
VAR_INPUT
	Enumeration : T_MAXSTRING;
	Value : ETcVnAdaptiveThresholdMethod;
END_VAR
AddEnumeration(Enumeration, Value);
END_METHOD

METHOD IsEnumeratorValueEqual : BOOL
VAR_INPUT
	Enumerator : I_KeyValueForwardEnumerator;
END_VAR
VAR
	storedValue : ETcVnAdaptiveThresholdMethod;
END_VAR
IF NOT Enumerator.TryGet(storedValue) THEN
	RETURN;
END_IF

IsEnumeratorValueEqual := storedValue = activeData;
END_METHOD

METHOD PUBLIC Clone : I_Datatype
VAR
    pClone : POINTER TO _ETcVnAdaptiveThresholdMethod;
END_VAR
pClone := __NEW(_ETcVnAdaptiveThresholdMethod(InitialValue := Value));
Clone := pClone^;
END_METHOD

PROPERTY PUBLIC Identifier : T_MAXSTRING
GET
Identifier := 'ETcVnAdaptiveThresholdMethod';
END_GET
END_PROPERTY

METHOD PUBLIC MakeReferenceTo
VAR_INPUT
	ReferenceTarget : REFERENCE TO ETcVnAdaptiveThresholdMethod;
END_VAR
activeData REF= ReferenceTarget;
SetBaseDatatypeReference();
END_METHOD

METHOD TryMakeReferenceTo : BOOL
VAR_INPUT
	Target : I_Datatype;
END_VAR
VAR
	targetAsEnum : I_EnumDatatype;
	pTargetData : POINTER TO ETcVnAdaptiveThresholdMethod;
END_VAR
IF NOT Target.TryResolveAsEnumDatatype(targetAsEnum) THEN
	RETURN;
END_IF

IF targetAsEnum.Identifier <> Identifier THEN
	RETURN;
END_IF

pTargetData := Target.Address;
activeData REF= pTargetData^;
SetBaseDatatypeReference();
TryMakeReferenceTo := TRUE;
END_METHOD

PROPERTY PUBLIC Value : ETcVnAdaptiveThresholdMethod
GET
Value := activeData;
END_GET
SET
activeData := Value;
END_SET
END_PROPERTY

END_FUNCTION_BLOCK

// Datatypes/Enums/_ETcVnBarcodeSearchDirection
{attribute 'linkalways'} 
{attribute 'no_explicit_call' := 'This FB is a CLASS and must be accessed using methods or properties'}
{attribute 'enable_dynamic_creation'}
FUNCTION_BLOCK _ETcVnBarcodeSearchDirection EXTENDS EnumDatatypeBase
VAR
	localData : ETcVnBarcodeSearchDirection;
	activeData : REFERENCE TO ETcVnBarcodeSearchDirection;
	enumBaseDatatype : _UDINT(localData);
END_VAR

METHOD PROTECTED SetBaseDatatypeReference
VAR_INPUT
END_VAR
enumBaseDatatype.MakeReferenceTo(activeData);
END_METHOD

PROPERTY PUBLIC Address : PVOID
GET
Address := ADR(activeData);
END_GET
END_PROPERTY

METHOD PUBLIC ClearReference
VAR_INPUT
END_VAR
activeData REF= localData;
SetBaseDatatypeReference();
END_METHOD

PROPERTY PUBLIC Size : UDINT
GET
Size := SIZEOF(activeData);
END_GET
END_PROPERTY

METHOD FB_init : BOOL
VAR_INPUT
	bInitRetains : BOOL; // if TRUE, the retain variables are initialized (warm start / cold start)
	bInCopyCode : BOOL;  // if TRUE, the instance afterwards gets moved into the copy code (online change)
	InitialValue : ETcVnBarcodeSearchDirection;
END_VAR
localData := InitialValue;
AddBaseDatatype(enumBaseDatatype);
ClearReference();

AddLocalEnumeration('TCVN_BSD_ANY', ETcVnBarcodeSearchDirection.TCVN_BSD_ANY);
AddLocalEnumeration('TCVN_BSD_HORIZONTAL', ETcVnBarcodeSearchDirection.TCVN_BSD_HORIZONTAL);
AddLocalEnumeration('TCVN_BSD_VERTICAL', ETcVnBarcodeSearchDirection.TCVN_BSD_VERTICAL);
END_METHOD

METHOD PRIVATE AddLocalEnumeration
VAR_INPUT
	Enumeration : T_MAXSTRING;
	Value : ETcVnBarcodeSearchDirection;
END_VAR
AddEnumeration(Enumeration, Value);
END_METHOD

METHOD IsEnumeratorValueEqual : BOOL
VAR_INPUT
	Enumerator : I_KeyValueForwardEnumerator;
END_VAR
VAR
	storedValue : ETcVnBarcodeSearchDirection;
END_VAR
IF NOT Enumerator.TryGet(storedValue) THEN
	RETURN;
END_IF

IsEnumeratorValueEqual := storedValue = activeData;
END_METHOD

METHOD PUBLIC Clone : I_Datatype
VAR
    pClone : POINTER TO _ETcVnBarcodeSearchDirection;
END_VAR
pClone := __NEW(_ETcVnBarcodeSearchDirection(InitialValue := Value));
Clone := pClone^;
END_METHOD

PROPERTY PUBLIC Identifier : T_MAXSTRING
GET
Identifier := 'ETcVnBarcodeSearchDirection';
END_GET
END_PROPERTY

METHOD PUBLIC MakeReferenceTo
VAR_INPUT
	ReferenceTarget : REFERENCE TO ETcVnBarcodeSearchDirection;
END_VAR
activeData REF= ReferenceTarget;
SetBaseDatatypeReference();
END_METHOD

METHOD TryMakeReferenceTo : BOOL
VAR_INPUT
	Target : I_Datatype;
END_VAR
VAR
	targetAsEnum : I_EnumDatatype;
	pTargetData : POINTER TO ETcVnBarcodeSearchDirection;
END_VAR
IF NOT Target.TryResolveAsEnumDatatype(targetAsEnum) THEN
	RETURN;
END_IF

IF targetAsEnum.Identifier <> Identifier THEN
	RETURN;
END_IF

pTargetData := Target.Address;
activeData REF= pTargetData^;
SetBaseDatatypeReference();
TryMakeReferenceTo := TRUE;
END_METHOD

PROPERTY PUBLIC Value : ETcVnBarcodeSearchDirection
GET
Value := activeData;
END_GET
SET
activeData := Value;
END_SET
END_PROPERTY

END_FUNCTION_BLOCK

// Datatypes/Enums/_ETcVnBarcodeType
{attribute 'linkalways'} 
{attribute 'no_explicit_call' := 'This FB is a CLASS and must be accessed using methods or properties'}
{attribute 'enable_dynamic_creation'}
FUNCTION_BLOCK _ETcVnBarcodeType EXTENDS EnumDatatypeBase
VAR
	localData : ETcVnBarcodeType;
	activeData : REFERENCE TO ETcVnBarcodeType;
	enumBaseDatatype : _UDINT(localData);
END_VAR

METHOD PROTECTED SetBaseDatatypeReference
VAR_INPUT
END_VAR
enumBaseDatatype.MakeReferenceTo(activeData);
END_METHOD

PROPERTY PUBLIC Address : PVOID
GET
Address := ADR(activeData);
END_GET
END_PROPERTY

METHOD PUBLIC ClearReference
VAR_INPUT
END_VAR
activeData REF= localData;
SetBaseDatatypeReference();
END_METHOD

PROPERTY PUBLIC Size : UDINT
GET
Size := SIZEOF(activeData);
END_GET
END_PROPERTY

METHOD FB_init : BOOL
VAR_INPUT
	bInitRetains : BOOL; // if TRUE, the retain variables are initialized (warm start / cold start)
	bInCopyCode : BOOL;  // if TRUE, the instance afterwards gets moved into the copy code (online change)
	InitialValue : ETcVnBarcodeType;
END_VAR
localData := InitialValue;
AddBaseDatatype(enumBaseDatatype);
ClearReference();

AddLocalEnumeration('TCVN_BT_CODABAR', ETcVnBarcodeType.TCVN_BT_CODABAR);
AddLocalEnumeration('TCVN_BT_CODE39', ETcVnBarcodeType.TCVN_BT_CODE39);
AddLocalEnumeration('TCVN_BT_CODE93', ETcVnBarcodeType.TCVN_BT_CODE93);
AddLocalEnumeration('TCVN_BT_CODE128', ETcVnBarcodeType.TCVN_BT_CODE128);
AddLocalEnumeration('TCVN_BT_EAN8', ETcVnBarcodeType.TCVN_BT_EAN8);
AddLocalEnumeration('TCVN_BT_EAN13', ETcVnBarcodeType.TCVN_BT_EAN13);
AddLocalEnumeration('TCVN_BT_ITF', ETcVnBarcodeType.TCVN_BT_ITF);
AddLocalEnumeration('TCVN_BT_UPCA', ETcVnBarcodeType.TCVN_BT_UPCA);
AddLocalEnumeration('TCVN_BT_UPCE', ETcVnBarcodeType.TCVN_BT_UPCE);
AddLocalEnumeration('TCVN_BT_ANY', ETcVnBarcodeType.TCVN_BT_ANY);
AddLocalEnumeration('TCVN_BT_CODE39EXTENDED', ETcVnBarcodeType.TCVN_BT_CODE39EXTENDED);
END_METHOD

METHOD PRIVATE AddLocalEnumeration
VAR_INPUT
	Enumeration : T_MAXSTRING;
	Value : ETcVnBarcodeType;
END_VAR
AddEnumeration(Enumeration, Value);
END_METHOD

METHOD IsEnumeratorValueEqual : BOOL
VAR_INPUT
	Enumerator : I_KeyValueForwardEnumerator;
END_VAR
VAR
	storedValue : ETcVnBarcodeType;
END_VAR
IF NOT Enumerator.TryGet(storedValue) THEN
	RETURN;
END_IF

IsEnumeratorValueEqual := storedValue = activeData;
END_METHOD

METHOD PUBLIC Clone : I_Datatype
VAR
    pClone : POINTER TO _ETcVnBarcodeType;
END_VAR
pClone := __NEW(_ETcVnBarcodeType(InitialValue := Value));
Clone := pClone^;
END_METHOD

PROPERTY PUBLIC Identifier : T_MAXSTRING
GET
Identifier := 'ETcVnBarcodeType';
END_GET
END_PROPERTY

METHOD PUBLIC MakeReferenceTo
VAR_INPUT
	ReferenceTarget : REFERENCE TO ETcVnBarcodeType;
END_VAR
activeData REF= ReferenceTarget;
SetBaseDatatypeReference();
END_METHOD

METHOD TryMakeReferenceTo : BOOL
VAR_INPUT
	Target : I_Datatype;
END_VAR
VAR
	targetAsEnum : I_EnumDatatype;
	pTargetData : POINTER TO ETcVnBarcodeType;
END_VAR
IF NOT Target.TryResolveAsEnumDatatype(targetAsEnum) THEN
	RETURN;
END_IF

IF targetAsEnum.Identifier <> Identifier THEN
	RETURN;
END_IF

pTargetData := Target.Address;
activeData REF= pTargetData^;
SetBaseDatatypeReference();
TryMakeReferenceTo := TRUE;
END_METHOD

PROPERTY PUBLIC Value : ETcVnBarcodeType
GET
Value := activeData;
END_GET
SET
activeData := Value;
END_SET
END_PROPERTY

END_FUNCTION_BLOCK

// Datatypes/Enums/_ETcVnBlobCombination
{attribute 'linkalways'} 
{attribute 'no_explicit_call' := 'This FB is a CLASS and must be accessed using methods or properties'}
{attribute 'enable_dynamic_creation'}
FUNCTION_BLOCK _ETcVnBlobCombination EXTENDS EnumDatatypeBase
VAR
	localData : ETcVnBlobCombination;
	activeData : REFERENCE TO ETcVnBlobCombination;
	enumBaseDatatype : _DINT(localData);
END_VAR

METHOD PROTECTED SetBaseDatatypeReference
VAR_INPUT
END_VAR
enumBaseDatatype.MakeReferenceTo(activeData);
END_METHOD

PROPERTY PUBLIC Address : PVOID
GET
Address := ADR(activeData);
END_GET
END_PROPERTY

METHOD PUBLIC ClearReference
VAR_INPUT
END_VAR
activeData REF= localData;
SetBaseDatatypeReference();
END_METHOD

PROPERTY PUBLIC Size : UDINT
GET
Size := SIZEOF(activeData);
END_GET
END_PROPERTY

METHOD FB_init : BOOL
VAR_INPUT
	bInitRetains : BOOL; // if TRUE, the retain variables are initialized (warm start / cold start)
	bInCopyCode : BOOL;  // if TRUE, the instance afterwards gets moved into the copy code (online change)
	InitialValue : ETcVnBlobCombination;
END_VAR
localData := InitialValue;
AddBaseDatatype(enumBaseDatatype);
ClearReference();

AddLocalEnumeration('TCVN_BC_SMALLEST', ETcVnBlobCombination.TCVN_BC_SMALLEST);
AddLocalEnumeration('TCVN_BC_LARGEST', ETcVnBlobCombination.TCVN_BC_LARGEST);
AddLocalEnumeration('TCVN_BC_MIN_THRESHOLD', ETcVnBlobCombination.TCVN_BC_MIN_THRESHOLD);
AddLocalEnumeration('TCVN_BC_MAX_THRESHOLD', ETcVnBlobCombination.TCVN_BC_MAX_THRESHOLD);
AddLocalEnumeration('TCVN_BC_MEDIAN_THRESHOLD', ETcVnBlobCombination.TCVN_BC_MEDIAN_THRESHOLD);
END_METHOD

METHOD PRIVATE AddLocalEnumeration
VAR_INPUT
	Enumeration : T_MAXSTRING;
	Value : ETcVnBlobCombination;
END_VAR
AddEnumeration(Enumeration, Value);
END_METHOD

METHOD IsEnumeratorValueEqual : BOOL
VAR_INPUT
	Enumerator : I_KeyValueForwardEnumerator;
END_VAR
VAR
	storedValue : ETcVnBlobCombination;
END_VAR
IF NOT Enumerator.TryGet(storedValue) THEN
	RETURN;
END_IF

IsEnumeratorValueEqual := storedValue = activeData;
END_METHOD

METHOD PUBLIC Clone : I_Datatype
VAR
    pClone : POINTER TO _ETcVnBlobCombination;
END_VAR
pClone := __NEW(_ETcVnBlobCombination(InitialValue := Value));
Clone := pClone^;
END_METHOD

PROPERTY PUBLIC Identifier : T_MAXSTRING
GET
Identifier := 'ETcVnBlobCombination';
END_GET
END_PROPERTY

METHOD PUBLIC MakeReferenceTo
VAR_INPUT
	ReferenceTarget : REFERENCE TO ETcVnBlobCombination;
END_VAR
activeData REF= ReferenceTarget;
SetBaseDatatypeReference();
END_METHOD

METHOD TryMakeReferenceTo : BOOL
VAR_INPUT
	Target : I_Datatype;
END_VAR
VAR
	targetAsEnum : I_EnumDatatype;
	pTargetData : POINTER TO ETcVnBlobCombination;
END_VAR
IF NOT Target.TryResolveAsEnumDatatype(targetAsEnum) THEN
	RETURN;
END_IF

IF targetAsEnum.Identifier <> Identifier THEN
	RETURN;
END_IF

pTargetData := Target.Address;
activeData REF= pTargetData^;
SetBaseDatatypeReference();
TryMakeReferenceTo := TRUE;
END_METHOD

PROPERTY PUBLIC Value : ETcVnBlobCombination
GET
Value := activeData;
END_GET
SET
activeData := Value;
END_SET
END_PROPERTY

END_FUNCTION_BLOCK

// Datatypes/Enums/_ETcVnBorderInterpolationMethod
{attribute 'linkalways'} 
{attribute 'no_explicit_call' := 'This FB is a CLASS and must be accessed using methods or properties'}
{attribute 'enable_dynamic_creation'}
FUNCTION_BLOCK _ETcVnBorderInterpolationMethod EXTENDS EnumDatatypeBase
VAR
	localData : ETcVnBorderInterpolationMethod;
	activeData : REFERENCE TO ETcVnBorderInterpolationMethod;
	enumBaseDatatype : _DINT(localData);
END_VAR

METHOD PROTECTED SetBaseDatatypeReference
VAR_INPUT
END_VAR
enumBaseDatatype.MakeReferenceTo(activeData);
END_METHOD

PROPERTY PUBLIC Address : PVOID
GET
Address := ADR(activeData);
END_GET
END_PROPERTY

METHOD PUBLIC ClearReference
VAR_INPUT
END_VAR
activeData REF= localData;
SetBaseDatatypeReference();
END_METHOD

PROPERTY PUBLIC Size : UDINT
GET
Size := SIZEOF(activeData);
END_GET
END_PROPERTY

METHOD FB_init : BOOL
VAR_INPUT
	bInitRetains : BOOL; // if TRUE, the retain variables are initialized (warm start / cold start)
	bInCopyCode : BOOL;  // if TRUE, the instance afterwards gets moved into the copy code (online change)
	InitialValue : ETcVnBorderInterpolationMethod;
END_VAR
localData := InitialValue;
AddBaseDatatype(enumBaseDatatype);
ClearReference();

AddLocalEnumeration('TCVN_BIM_CONSTANT', ETcVnBorderInterpolationMethod.TCVN_BIM_CONSTANT);
AddLocalEnumeration('TCVN_BIM_REPLICATE', ETcVnBorderInterpolationMethod.TCVN_BIM_REPLICATE);
AddLocalEnumeration('TCVN_BIM_REFLECT', ETcVnBorderInterpolationMethod.TCVN_BIM_REFLECT);
AddLocalEnumeration('TCVN_BIM_WRAP', ETcVnBorderInterpolationMethod.TCVN_BIM_WRAP);
AddLocalEnumeration('TCVN_BIM_REFLECT_101', ETcVnBorderInterpolationMethod.TCVN_BIM_REFLECT_101);
AddLocalEnumeration('TCVN_BIM_DEFAULT', ETcVnBorderInterpolationMethod.TCVN_BIM_DEFAULT);
AddLocalEnumeration('TCVN_BIM_TRANSPARENT', ETcVnBorderInterpolationMethod.TCVN_BIM_TRANSPARENT);
AddLocalEnumeration('TCVN_BIM_ISOLATED_CONSTANT', ETcVnBorderInterpolationMethod.TCVN_BIM_ISOLATED_CONSTANT);
AddLocalEnumeration('TCVN_BIM_ISOLATED_REPLICATE', ETcVnBorderInterpolationMethod.TCVN_BIM_ISOLATED_REPLICATE);
AddLocalEnumeration('TCVN_BIM_ISOLATED_REFLECT', ETcVnBorderInterpolationMethod.TCVN_BIM_ISOLATED_REFLECT);
AddLocalEnumeration('TCVN_BIM_ISOLATED_WRAP', ETcVnBorderInterpolationMethod.TCVN_BIM_ISOLATED_WRAP);
AddLocalEnumeration('TCVN_BIM_ISOLATED_REFLECT_101', ETcVnBorderInterpolationMethod.TCVN_BIM_ISOLATED_REFLECT_101);
END_METHOD

METHOD PRIVATE AddLocalEnumeration
VAR_INPUT
	Enumeration : T_MAXSTRING;
	Value : ETcVnBorderInterpolationMethod;
END_VAR
AddEnumeration(Enumeration, Value);
END_METHOD

METHOD IsEnumeratorValueEqual : BOOL
VAR_INPUT
	Enumerator : I_KeyValueForwardEnumerator;
END_VAR
VAR
	storedValue : ETcVnBorderInterpolationMethod;
END_VAR
IF NOT Enumerator.TryGet(storedValue) THEN
	RETURN;
END_IF

IsEnumeratorValueEqual := storedValue = activeData;
END_METHOD

METHOD PUBLIC Clone : I_Datatype
VAR
    pClone : POINTER TO _ETcVnBorderInterpolationMethod;
END_VAR
pClone := __NEW(_ETcVnBorderInterpolationMethod(InitialValue := Value));
Clone := pClone^;
END_METHOD

PROPERTY PUBLIC Identifier : T_MAXSTRING
GET
Identifier := 'ETcVnBorderInterpolationMethod';
END_GET
END_PROPERTY

METHOD PUBLIC MakeReferenceTo
VAR_INPUT
	ReferenceTarget : REFERENCE TO ETcVnBorderInterpolationMethod;
END_VAR
activeData REF= ReferenceTarget;
SetBaseDatatypeReference();
END_METHOD

METHOD TryMakeReferenceTo : BOOL
VAR_INPUT
	Target : I_Datatype;
END_VAR
VAR
	targetAsEnum : I_EnumDatatype;
	pTargetData : POINTER TO ETcVnBorderInterpolationMethod;
END_VAR
IF NOT Target.TryResolveAsEnumDatatype(targetAsEnum) THEN
	RETURN;
END_IF

IF targetAsEnum.Identifier <> Identifier THEN
	RETURN;
END_IF

pTargetData := Target.Address;
activeData REF= pTargetData^;
SetBaseDatatypeReference();
TryMakeReferenceTo := TRUE;
END_METHOD

PROPERTY PUBLIC Value : ETcVnBorderInterpolationMethod
GET
Value := activeData;
END_GET
SET
activeData := Value;
END_SET
END_PROPERTY

END_FUNCTION_BLOCK

// Datatypes/Enums/_ETcVnCalibrationPattern
{attribute 'linkalways'} 
{attribute 'no_explicit_call' := 'This FB is a CLASS and must be accessed using methods or properties'}
{attribute 'enable_dynamic_creation'}
FUNCTION_BLOCK _ETcVnCalibrationPattern EXTENDS EnumDatatypeBase
VAR
	localData : ETcVnCalibrationPattern;
	activeData : REFERENCE TO ETcVnCalibrationPattern;
	enumBaseDatatype : _DINT(localData);
END_VAR

METHOD PROTECTED SetBaseDatatypeReference
VAR_INPUT
END_VAR
enumBaseDatatype.MakeReferenceTo(activeData);
END_METHOD

PROPERTY PUBLIC Address : PVOID
GET
Address := ADR(activeData);
END_GET
END_PROPERTY

METHOD PUBLIC ClearReference
VAR_INPUT
END_VAR
activeData REF= localData;
SetBaseDatatypeReference();
END_METHOD

PROPERTY PUBLIC Size : UDINT
GET
Size := SIZEOF(activeData);
END_GET
END_PROPERTY

METHOD FB_init : BOOL
VAR_INPUT
	bInitRetains : BOOL; // if TRUE, the retain variables are initialized (warm start / cold start)
	bInCopyCode : BOOL;  // if TRUE, the instance afterwards gets moved into the copy code (online change)
	InitialValue : ETcVnCalibrationPattern;
END_VAR
localData := InitialValue;
AddBaseDatatype(enumBaseDatatype);
ClearReference();

AddLocalEnumeration('TCVN_CP_CIRCLES_SYM', ETcVnCalibrationPattern.TCVN_CP_CIRCLES_SYM);
AddLocalEnumeration('TCVN_CP_CIRCLES_ASYM', ETcVnCalibrationPattern.TCVN_CP_CIRCLES_ASYM);
AddLocalEnumeration('TCVN_CP_CIRCLES_ASYM_INDENT', ETcVnCalibrationPattern.TCVN_CP_CIRCLES_ASYM_INDENT);
END_METHOD

METHOD PRIVATE AddLocalEnumeration
VAR_INPUT
	Enumeration : T_MAXSTRING;
	Value : ETcVnCalibrationPattern;
END_VAR
AddEnumeration(Enumeration, Value);
END_METHOD

METHOD IsEnumeratorValueEqual : BOOL
VAR_INPUT
	Enumerator : I_KeyValueForwardEnumerator;
END_VAR
VAR
	storedValue : ETcVnCalibrationPattern;
END_VAR
IF NOT Enumerator.TryGet(storedValue) THEN
	RETURN;
END_IF

IsEnumeratorValueEqual := storedValue = activeData;
END_METHOD

METHOD PUBLIC Clone : I_Datatype
VAR
    pClone : POINTER TO _ETcVnCalibrationPattern;
END_VAR
pClone := __NEW(_ETcVnCalibrationPattern(InitialValue := Value));
Clone := pClone^;
END_METHOD

PROPERTY PUBLIC Identifier : T_MAXSTRING
GET
Identifier := 'ETcVnCalibrationPattern';
END_GET
END_PROPERTY

METHOD PUBLIC MakeReferenceTo
VAR_INPUT
	ReferenceTarget : REFERENCE TO ETcVnCalibrationPattern;
END_VAR
activeData REF= ReferenceTarget;
SetBaseDatatypeReference();
END_METHOD

METHOD TryMakeReferenceTo : BOOL
VAR_INPUT
	Target : I_Datatype;
END_VAR
VAR
	targetAsEnum : I_EnumDatatype;
	pTargetData : POINTER TO ETcVnCalibrationPattern;
END_VAR
IF NOT Target.TryResolveAsEnumDatatype(targetAsEnum) THEN
	RETURN;
END_IF

IF targetAsEnum.Identifier <> Identifier THEN
	RETURN;
END_IF

pTargetData := Target.Address;
activeData REF= pTargetData^;
SetBaseDatatypeReference();
TryMakeReferenceTo := TRUE;
END_METHOD

PROPERTY PUBLIC Value : ETcVnCalibrationPattern
GET
Value := activeData;
END_GET
SET
activeData := Value;
END_SET
END_PROPERTY

END_FUNCTION_BLOCK

// Datatypes/Enums/_ETcVnCalibrationPatternOrigin
{attribute 'linkalways'} 
{attribute 'no_explicit_call' := 'This FB is a CLASS and must be accessed using methods or properties'}
{attribute 'enable_dynamic_creation'}
FUNCTION_BLOCK _ETcVnCalibrationPatternOrigin EXTENDS EnumDatatypeBase
VAR
	localData : ETcVnCalibrationPatternOrigin;
	activeData : REFERENCE TO ETcVnCalibrationPatternOrigin;
	enumBaseDatatype : _DINT(localData);
END_VAR

METHOD PROTECTED SetBaseDatatypeReference
VAR_INPUT
END_VAR
enumBaseDatatype.MakeReferenceTo(activeData);
END_METHOD

PROPERTY PUBLIC Address : PVOID
GET
Address := ADR(activeData);
END_GET
END_PROPERTY

METHOD PUBLIC ClearReference
VAR_INPUT
END_VAR
activeData REF= localData;
SetBaseDatatypeReference();
END_METHOD

PROPERTY PUBLIC Size : UDINT
GET
Size := SIZEOF(activeData);
END_GET
END_PROPERTY

METHOD FB_init : BOOL
VAR_INPUT
	bInitRetains : BOOL; // if TRUE, the retain variables are initialized (warm start / cold start)
	bInCopyCode : BOOL;  // if TRUE, the instance afterwards gets moved into the copy code (online change)
	InitialValue : ETcVnCalibrationPatternOrigin;
END_VAR
localData := InitialValue;
AddBaseDatatype(enumBaseDatatype);
ClearReference();

AddLocalEnumeration('TCVN_CPO_TOPLEFT', ETcVnCalibrationPatternOrigin.TCVN_CPO_TOPLEFT);
AddLocalEnumeration('TCVN_CPO_TOPCENTER', ETcVnCalibrationPatternOrigin.TCVN_CPO_TOPCENTER);
AddLocalEnumeration('TCVN_CPO_TOPRIGHT', ETcVnCalibrationPatternOrigin.TCVN_CPO_TOPRIGHT);
AddLocalEnumeration('TCVN_CPO_CENTERLEFT', ETcVnCalibrationPatternOrigin.TCVN_CPO_CENTERLEFT);
AddLocalEnumeration('TCVN_CPO_CENTER', ETcVnCalibrationPatternOrigin.TCVN_CPO_CENTER);
AddLocalEnumeration('TCVN_CPO_CENTERRIGHT', ETcVnCalibrationPatternOrigin.TCVN_CPO_CENTERRIGHT);
AddLocalEnumeration('TCVN_CPO_BOTTOMLEFT', ETcVnCalibrationPatternOrigin.TCVN_CPO_BOTTOMLEFT);
AddLocalEnumeration('TCVN_CPO_BOTTOMCENTER', ETcVnCalibrationPatternOrigin.TCVN_CPO_BOTTOMCENTER);
AddLocalEnumeration('TCVN_CPO_BOTTOMRIGHT', ETcVnCalibrationPatternOrigin.TCVN_CPO_BOTTOMRIGHT);
END_METHOD

METHOD PRIVATE AddLocalEnumeration
VAR_INPUT
	Enumeration : T_MAXSTRING;
	Value : ETcVnCalibrationPatternOrigin;
END_VAR
AddEnumeration(Enumeration, Value);
END_METHOD

METHOD IsEnumeratorValueEqual : BOOL
VAR_INPUT
	Enumerator : I_KeyValueForwardEnumerator;
END_VAR
VAR
	storedValue : ETcVnCalibrationPatternOrigin;
END_VAR
IF NOT Enumerator.TryGet(storedValue) THEN
	RETURN;
END_IF

IsEnumeratorValueEqual := storedValue = activeData;
END_METHOD

METHOD PUBLIC Clone : I_Datatype
VAR
    pClone : POINTER TO _ETcVnCalibrationPatternOrigin;
END_VAR
pClone := __NEW(_ETcVnCalibrationPatternOrigin(InitialValue := Value));
Clone := pClone^;
END_METHOD

PROPERTY PUBLIC Identifier : T_MAXSTRING
GET
Identifier := 'ETcVnCalibrationPatternOrigin';
END_GET
END_PROPERTY

METHOD PUBLIC MakeReferenceTo
VAR_INPUT
	ReferenceTarget : REFERENCE TO ETcVnCalibrationPatternOrigin;
END_VAR
activeData REF= ReferenceTarget;
SetBaseDatatypeReference();
END_METHOD

METHOD TryMakeReferenceTo : BOOL
VAR_INPUT
	Target : I_Datatype;
END_VAR
VAR
	targetAsEnum : I_EnumDatatype;
	pTargetData : POINTER TO ETcVnCalibrationPatternOrigin;
END_VAR
IF NOT Target.TryResolveAsEnumDatatype(targetAsEnum) THEN
	RETURN;
END_IF

IF targetAsEnum.Identifier <> Identifier THEN
	RETURN;
END_IF

pTargetData := Target.Address;
activeData REF= pTargetData^;
SetBaseDatatypeReference();
TryMakeReferenceTo := TRUE;
END_METHOD

PROPERTY PUBLIC Value : ETcVnCalibrationPatternOrigin
GET
Value := activeData;
END_GET
SET
activeData := Value;
END_SET
END_PROPERTY

END_FUNCTION_BLOCK

// Datatypes/Enums/_ETcVnCameraState
{attribute 'linkalways'} 
{attribute 'no_explicit_call' := 'This FB is a CLASS and must be accessed using methods or properties'}
{attribute 'enable_dynamic_creation'}
FUNCTION_BLOCK _ETcVnCameraState EXTENDS EnumDatatypeBase
VAR
	localData : ETcVnCameraState;
	activeData : REFERENCE TO ETcVnCameraState;
	enumBaseDatatype : _DINT(localData);
END_VAR

METHOD PROTECTED SetBaseDatatypeReference
VAR_INPUT
END_VAR
enumBaseDatatype.MakeReferenceTo(activeData);
END_METHOD

PROPERTY PUBLIC Address : PVOID
GET
Address := ADR(activeData);
END_GET
END_PROPERTY

METHOD PUBLIC ClearReference
VAR_INPUT
END_VAR
activeData REF= localData;
SetBaseDatatypeReference();
END_METHOD

PROPERTY PUBLIC Size : UDINT
GET
Size := SIZEOF(activeData);
END_GET
END_PROPERTY

METHOD FB_init : BOOL
VAR_INPUT
	bInitRetains : BOOL; // if TRUE, the retain variables are initialized (warm start / cold start)
	bInCopyCode : BOOL;  // if TRUE, the instance afterwards gets moved into the copy code (online change)
	InitialValue : ETcVnCameraState;
END_VAR
localData := InitialValue;
AddBaseDatatype(enumBaseDatatype);
ClearReference();

AddLocalEnumeration('TCVN_CS_ERROR', ETcVnCameraState.TCVN_CS_ERROR);
AddLocalEnumeration('TCVN_CS_INITIAL', ETcVnCameraState.TCVN_CS_INITIAL);
AddLocalEnumeration('TCVN_CS_INITIALIZING', ETcVnCameraState.TCVN_CS_INITIALIZING);
AddLocalEnumeration('TCVN_CS_INITIALIZED', ETcVnCameraState.TCVN_CS_INITIALIZED);
AddLocalEnumeration('TCVN_CS_OPENING', ETcVnCameraState.TCVN_CS_OPENING);
AddLocalEnumeration('TCVN_CS_OPENED', ETcVnCameraState.TCVN_CS_OPENED);
AddLocalEnumeration('TCVN_CS_STARTACQUISITION', ETcVnCameraState.TCVN_CS_STARTACQUISITION);
AddLocalEnumeration('TCVN_CS_ACQUIRING', ETcVnCameraState.TCVN_CS_ACQUIRING);
AddLocalEnumeration('TCVN_CS_STOPACQUISITION', ETcVnCameraState.TCVN_CS_STOPACQUISITION);
AddLocalEnumeration('TCVN_CS_RESETTINGFEATURES', ETcVnCameraState.TCVN_CS_RESETTINGFEATURES);
AddLocalEnumeration('TCVN_CS_TRIGGERING', ETcVnCameraState.TCVN_CS_TRIGGERING);
AddLocalEnumeration('TCVN_CS_CLOSING', ETcVnCameraState.TCVN_CS_CLOSING);
END_METHOD

METHOD PRIVATE AddLocalEnumeration
VAR_INPUT
	Enumeration : T_MAXSTRING;
	Value : ETcVnCameraState;
END_VAR
AddEnumeration(Enumeration, Value);
END_METHOD

METHOD IsEnumeratorValueEqual : BOOL
VAR_INPUT
	Enumerator : I_KeyValueForwardEnumerator;
END_VAR
VAR
	storedValue : ETcVnCameraState;
END_VAR
IF NOT Enumerator.TryGet(storedValue) THEN
	RETURN;
END_IF

IsEnumeratorValueEqual := storedValue = activeData;
END_METHOD

METHOD PUBLIC Clone : I_Datatype
VAR
    pClone : POINTER TO _ETcVnCameraState;
END_VAR
pClone := __NEW(_ETcVnCameraState(InitialValue := Value));
Clone := pClone^;
END_METHOD

PROPERTY PUBLIC Identifier : T_MAXSTRING
GET
Identifier := 'ETcVnCameraState';
END_GET
END_PROPERTY

METHOD PUBLIC MakeReferenceTo
VAR_INPUT
	ReferenceTarget : REFERENCE TO ETcVnCalibrationPatternOrigin;
END_VAR
activeData REF= ReferenceTarget;
SetBaseDatatypeReference();
END_METHOD

METHOD TryMakeReferenceTo : BOOL
VAR_INPUT
	Target : I_Datatype;
END_VAR
VAR
	targetAsEnum : I_EnumDatatype;
	pTargetData : POINTER TO ETcVnCameraState;
END_VAR
IF NOT Target.TryResolveAsEnumDatatype(targetAsEnum) THEN
	RETURN;
END_IF

IF targetAsEnum.Identifier <> Identifier THEN
	RETURN;
END_IF

pTargetData := Target.Address;
activeData REF= pTargetData^;
SetBaseDatatypeReference();
TryMakeReferenceTo := TRUE;
END_METHOD

PROPERTY PUBLIC Value : ETcVnCameraState
GET
Value := activeData;
END_GET
SET
activeData := Value;
END_SET
END_PROPERTY

END_FUNCTION_BLOCK

// Datatypes/Enums/_ETcVnClusteringAlgorithm
{attribute 'linkalways'} 
{attribute 'no_explicit_call' := 'This FB is a CLASS and must be accessed using methods or properties'}
{attribute 'enable_dynamic_creation'}
FUNCTION_BLOCK _ETcVnClusteringAlgorithm EXTENDS EnumDatatypeBase
VAR
	localData : ETcVnClusteringAlgorithm;
	activeData : REFERENCE TO ETcVnClusteringAlgorithm;
	enumBaseDatatype : _DINT(localData);
END_VAR

METHOD PROTECTED SetBaseDatatypeReference
VAR_INPUT
END_VAR
enumBaseDatatype.MakeReferenceTo(activeData);
END_METHOD

PROPERTY PUBLIC Address : PVOID
GET
Address := ADR(activeData);
END_GET
END_PROPERTY

METHOD PUBLIC ClearReference
VAR_INPUT
END_VAR
activeData REF= localData;
SetBaseDatatypeReference();
END_METHOD

PROPERTY PUBLIC Size : UDINT
GET
Size := SIZEOF(activeData);
END_GET
END_PROPERTY

METHOD FB_init : BOOL
VAR_INPUT
	bInitRetains : BOOL; // if TRUE, the retain variables are initialized (warm start / cold start)
	bInCopyCode : BOOL;  // if TRUE, the instance afterwards gets moved into the copy code (online change)
	InitialValue : ETcVnClusteringAlgorithm;
END_VAR
localData := InitialValue;
AddBaseDatatype(enumBaseDatatype);
ClearReference();

AddLocalEnumeration('TCVN_CA_KMEANSPP', ETcVnClusteringAlgorithm.TCVN_CA_KMEANSPP);
AddLocalEnumeration('TCVN_CA_LBG', ETcVnClusteringAlgorithm.TCVN_CA_LBG);
END_METHOD

METHOD PRIVATE AddLocalEnumeration
VAR_INPUT
	Enumeration : T_MAXSTRING;
	Value : ETcVnClusteringAlgorithm;
END_VAR
AddEnumeration(Enumeration, Value);
END_METHOD

METHOD IsEnumeratorValueEqual : BOOL
VAR_INPUT
	Enumerator : I_KeyValueForwardEnumerator;
END_VAR
VAR
	storedValue : ETcVnClusteringAlgorithm;
END_VAR
IF NOT Enumerator.TryGet(storedValue) THEN
	RETURN;
END_IF

IsEnumeratorValueEqual := storedValue = activeData;
END_METHOD

METHOD PUBLIC Clone : I_Datatype
VAR
    pClone : POINTER TO _ETcVnClusteringAlgorithm;
END_VAR
pClone := __NEW(_ETcVnClusteringAlgorithm(InitialValue := Value));
Clone := pClone^;
END_METHOD

PROPERTY PUBLIC Identifier : T_MAXSTRING
GET
Identifier := 'ETcVnClusteringAlgorithm';
END_GET
END_PROPERTY

METHOD PUBLIC MakeReferenceTo
VAR_INPUT
	ReferenceTarget : REFERENCE TO ETcVnCalibrationPatternOrigin;
END_VAR
activeData REF= ReferenceTarget;
SetBaseDatatypeReference();
END_METHOD

METHOD TryMakeReferenceTo : BOOL
VAR_INPUT
	Target : I_Datatype;
END_VAR
VAR
	targetAsEnum : I_EnumDatatype;
	pTargetData : POINTER TO ETcVnClusteringAlgorithm;
END_VAR
IF NOT Target.TryResolveAsEnumDatatype(targetAsEnum) THEN
	RETURN;
END_IF

IF targetAsEnum.Identifier <> Identifier THEN
	RETURN;
END_IF

pTargetData := Target.Address;
activeData REF= pTargetData^;
SetBaseDatatypeReference();
TryMakeReferenceTo := TRUE;
END_METHOD

PROPERTY PUBLIC Value : ETcVnClusteringAlgorithm
GET
Value := activeData;
END_GET
SET
activeData := Value;
END_SET
END_PROPERTY

END_FUNCTION_BLOCK

// Datatypes/Enums/_ETcVnColorMap
{attribute 'linkalways'} 
{attribute 'no_explicit_call' := 'This FB is a CLASS and must be accessed using methods or properties'}
{attribute 'enable_dynamic_creation'}
FUNCTION_BLOCK _ETcVnColorMap EXTENDS EnumDatatypeBase
VAR
	localData : ETcVnColorMap;
	activeData : REFERENCE TO ETcVnColorMap;
	enumBaseDatatype : _DINT(localData);
END_VAR

METHOD PROTECTED SetBaseDatatypeReference
VAR_INPUT
END_VAR
enumBaseDatatype.MakeReferenceTo(activeData);
END_METHOD

PROPERTY PUBLIC Address : PVOID
GET
Address := ADR(activeData);
END_GET
END_PROPERTY

METHOD PUBLIC ClearReference
VAR_INPUT
END_VAR
activeData REF= localData;
SetBaseDatatypeReference();
END_METHOD

PROPERTY PUBLIC Size : UDINT
GET
Size := SIZEOF(activeData);
END_GET
END_PROPERTY

METHOD FB_init : BOOL
VAR_INPUT
	bInitRetains : BOOL; // if TRUE, the retain variables are initialized (warm start / cold start)
	bInCopyCode : BOOL;  // if TRUE, the instance afterwards gets moved into the copy code (online change)
	InitialValue : ETcVnColorMap;
END_VAR
localData := InitialValue;
AddBaseDatatype(enumBaseDatatype);
ClearReference();

AddLocalEnumeration('TCVN_CM_AUTUMN', ETcVnColorMap.TCVN_CM_AUTUMN);
AddLocalEnumeration('TCVN_CM_BONE', ETcVnColorMap.TCVN_CM_BONE);
AddLocalEnumeration('TCVN_CM_JET', ETcVnColorMap.TCVN_CM_JET);
AddLocalEnumeration('TCVN_CM_WINTER', ETcVnColorMap.TCVN_CM_WINTER);
AddLocalEnumeration('TCVN_CM_RAINBOW', ETcVnColorMap.TCVN_CM_RAINBOW);
AddLocalEnumeration('TCVN_CM_OCEAN', ETcVnColorMap.TCVN_CM_OCEAN);
AddLocalEnumeration('TCVN_CM_SUMMER', ETcVnColorMap.TCVN_CM_SUMMER);
AddLocalEnumeration('TCVN_CM_SPRING', ETcVnColorMap.TCVN_CM_SPRING);
AddLocalEnumeration('TCVN_CM_COOL', ETcVnColorMap.TCVN_CM_COOL);
AddLocalEnumeration('TCVN_CM_HSV', ETcVnColorMap.TCVN_CM_HSV);
AddLocalEnumeration('TCVN_CM_PINK', ETcVnColorMap.TCVN_CM_PINK);
AddLocalEnumeration('TCVN_CM_HOT', ETcVnColorMap.TCVN_CM_HOT);
AddLocalEnumeration('TCVN_CM_PARULA', ETcVnColorMap.TCVN_CM_PARULA);
AddLocalEnumeration('TCVN_CM_MAGMA', ETcVnColorMap.TCVN_CM_MAGMA);
AddLocalEnumeration('TCVN_CM_INFERNO', ETcVnColorMap.TCVN_CM_INFERNO);
AddLocalEnumeration('TCVN_CM_PLASMA', ETcVnColorMap.TCVN_CM_PLASMA);
AddLocalEnumeration('TCVN_CM_VIRIDIS', ETcVnColorMap.TCVN_CM_VIRIDIS);
AddLocalEnumeration('TCVN_CM_CIVIDIS', ETcVnColorMap.TCVN_CM_CIVIDIS);
AddLocalEnumeration('TCVN_CM_TWILIGHT', ETcVnColorMap.TCVN_CM_TWILIGHT);
AddLocalEnumeration('TCVN_CM_TWILIGHT_SHIFTED', ETcVnColorMap.TCVN_CM_TWILIGHT_SHIFTED);
AddLocalEnumeration('TCVN_CM_TURBO', ETcVnColorMap.TCVN_CM_TURBO);
END_METHOD

METHOD PRIVATE AddLocalEnumeration
VAR_INPUT
	Enumeration : T_MAXSTRING;
	Value : ETcVnColorMap;
END_VAR
AddEnumeration(Enumeration, Value);
END_METHOD

METHOD IsEnumeratorValueEqual : BOOL
VAR_INPUT
	Enumerator : I_KeyValueForwardEnumerator;
END_VAR
VAR
	storedValue : ETcVnColorMap;
END_VAR
IF NOT Enumerator.TryGet(storedValue) THEN
	RETURN;
END_IF

IsEnumeratorValueEqual := storedValue = activeData;
END_METHOD

METHOD PUBLIC Clone : I_Datatype
VAR
    pClone : POINTER TO _ETcVnColorMap;
END_VAR
pClone := __NEW(_ETcVnColorMap(InitialValue := Value));
Clone := pClone^;
END_METHOD

PROPERTY PUBLIC Identifier : T_MAXSTRING
GET
Identifier := 'ETcVnColorMap';
END_GET
END_PROPERTY

METHOD PUBLIC MakeReferenceTo
VAR_INPUT
	ReferenceTarget : REFERENCE TO ETcVnCalibrationPatternOrigin;
END_VAR
activeData REF= ReferenceTarget;
SetBaseDatatypeReference();
END_METHOD

METHOD TryMakeReferenceTo : BOOL
VAR_INPUT
	Target : I_Datatype;
END_VAR
VAR
	targetAsEnum : I_EnumDatatype;
	pTargetData : POINTER TO ETcVnColorMap;
END_VAR
IF NOT Target.TryResolveAsEnumDatatype(targetAsEnum) THEN
	RETURN;
END_IF

IF targetAsEnum.Identifier <> Identifier THEN
	RETURN;
END_IF

pTargetData := Target.Address;
activeData REF= pTargetData^;
SetBaseDatatypeReference();
TryMakeReferenceTo := TRUE;
END_METHOD

PROPERTY PUBLIC Value : ETcVnColorMap
GET
Value := activeData;
END_GET
SET
activeData := Value;
END_SET
END_PROPERTY

END_FUNCTION_BLOCK

// Datatypes/Enums/_ETcVnColorMapSize
{attribute 'linkalways'} 
{attribute 'no_explicit_call' := 'This FB is a CLASS and must be accessed using methods or properties'}
{attribute 'enable_dynamic_creation'}
FUNCTION_BLOCK _ETcVnColorMapSize EXTENDS EnumDatatypeBase
VAR
	localData : ETcVnColorMapSize;
	activeData : REFERENCE TO ETcVnColorMapSize;
	enumBaseDatatype : _UDINT(localData);
END_VAR

METHOD PROTECTED SetBaseDatatypeReference
VAR_INPUT
END_VAR
enumBaseDatatype.MakeReferenceTo(activeData);
END_METHOD

PROPERTY PUBLIC Address : PVOID
GET
Address := ADR(activeData);
END_GET
END_PROPERTY

METHOD PUBLIC ClearReference
VAR_INPUT
END_VAR
activeData REF= localData;
SetBaseDatatypeReference();
END_METHOD

PROPERTY PUBLIC Size : UDINT
GET
Size := SIZEOF(activeData);
END_GET
END_PROPERTY

METHOD FB_init : BOOL
VAR_INPUT
	bInitRetains : BOOL; // if TRUE, the retain variables are initialized (warm start / cold start)
	bInCopyCode : BOOL;  // if TRUE, the instance afterwards gets moved into the copy code (online change)
	InitialValue : ETcVnColorMapSize;
END_VAR
localData := InitialValue;
AddBaseDatatype(enumBaseDatatype);
ClearReference();

AddLocalEnumeration('TCVN_CMS_256', ETcVnColorMapSize.TCVN_CMS_256);
AddLocalEnumeration('TCVN_CMS_65536', ETcVnColorMapSize.TCVN_CMS_65536);
END_METHOD

METHOD PRIVATE AddLocalEnumeration
VAR_INPUT
	Enumeration : T_MAXSTRING;
	Value : ETcVnColorMapSize;
END_VAR
AddEnumeration(Enumeration, Value);
END_METHOD

METHOD IsEnumeratorValueEqual : BOOL
VAR_INPUT
	Enumerator : I_KeyValueForwardEnumerator;
END_VAR
VAR
	storedValue : ETcVnColorMapSize;
END_VAR
IF NOT Enumerator.TryGet(storedValue) THEN
	RETURN;
END_IF

IsEnumeratorValueEqual := storedValue = activeData;
END_METHOD

METHOD PUBLIC Clone : I_Datatype
VAR
    pClone : POINTER TO _ETcVnColorMapSize;
END_VAR
pClone := __NEW(_ETcVnColorMapSize(InitialValue := Value));
Clone := pClone^;
END_METHOD

PROPERTY PUBLIC Identifier : T_MAXSTRING
GET
Identifier := 'ETcVnColorMapSize';
END_GET
END_PROPERTY

METHOD PUBLIC MakeReferenceTo
VAR_INPUT
	ReferenceTarget : REFERENCE TO ETcVnColorMapSize;
END_VAR
activeData REF= ReferenceTarget;
SetBaseDatatypeReference();
END_METHOD

METHOD TryMakeReferenceTo : BOOL
VAR_INPUT
	Target : I_Datatype;
END_VAR
VAR
	targetAsEnum : I_EnumDatatype;
	pTargetData : POINTER TO ETcVnColorMapSize;
END_VAR
IF NOT Target.TryResolveAsEnumDatatype(targetAsEnum) THEN
	RETURN;
END_IF

IF targetAsEnum.Identifier <> Identifier THEN
	RETURN;
END_IF

pTargetData := Target.Address;
activeData REF= pTargetData^;
SetBaseDatatypeReference();
TryMakeReferenceTo := TRUE;
END_METHOD

PROPERTY PUBLIC Value : ETcVnColorMapSize
GET
Value := activeData;
END_GET
SET
activeData := Value;
END_SET
END_PROPERTY

END_FUNCTION_BLOCK

// Datatypes/Enums/_ETcVnColorSpaceTransform
{attribute 'linkalways'} 
{attribute 'no_explicit_call' := 'This FB is a CLASS and must be accessed using methods or properties'}
{attribute 'enable_dynamic_creation'}
FUNCTION_BLOCK _ETcVnColorSpaceTransform EXTENDS EnumDatatypeBase
VAR
	localData : ETcVnColorSpaceTransform;
	activeData : REFERENCE TO ETcVnColorSpaceTransform;
	enumBaseDatatype : _DINT(localData);
END_VAR

METHOD PROTECTED SetBaseDatatypeReference
VAR_INPUT
END_VAR
enumBaseDatatype.MakeReferenceTo(activeData);
END_METHOD

PROPERTY PUBLIC Address : PVOID
GET
Address := ADR(activeData);
END_GET
END_PROPERTY

METHOD PUBLIC ClearReference
VAR_INPUT
END_VAR
activeData REF= localData;
SetBaseDatatypeReference();
END_METHOD

PROPERTY PUBLIC Size : UDINT
GET
Size := SIZEOF(activeData);
END_GET
END_PROPERTY

METHOD FB_init : BOOL
VAR_INPUT
	bInitRetains : BOOL; // if TRUE, the retain variables are initialized (warm start / cold start)
	bInCopyCode : BOOL;  // if TRUE, the instance afterwards gets moved into the copy code (online change)
	InitialValue : ETcVnColorSpaceTransform;
END_VAR
localData := InitialValue;
AddBaseDatatype(enumBaseDatatype);
ClearReference();

AddLocalEnumeration('TCVN_CST_BGR_TO_BGRA', ETcVnColorSpaceTransform.TCVN_CST_BGR_TO_BGRA);
AddLocalEnumeration('TCVN_CST_RGB_TO_RGBA', ETcVnColorSpaceTransform.TCVN_CST_RGB_TO_RGBA);
AddLocalEnumeration('TCVN_CST_BGRA_TO_BGR', ETcVnColorSpaceTransform.TCVN_CST_BGRA_TO_BGR);
AddLocalEnumeration('TCVN_CST_RGBA_TO_RGB', ETcVnColorSpaceTransform.TCVN_CST_RGBA_TO_RGB);
AddLocalEnumeration('TCVN_CST_BGR_TO_RGBA', ETcVnColorSpaceTransform.TCVN_CST_BGR_TO_RGBA);
AddLocalEnumeration('TCVN_CST_RGB_TO_BGRA', ETcVnColorSpaceTransform.TCVN_CST_RGB_TO_BGRA);
AddLocalEnumeration('TCVN_CST_BGRA_TO_RGB', ETcVnColorSpaceTransform.TCVN_CST_BGRA_TO_RGB);
AddLocalEnumeration('TCVN_CST_RGBA_TO_BGR', ETcVnColorSpaceTransform.TCVN_CST_RGBA_TO_BGR);
AddLocalEnumeration('TCVN_CST_BGR_TO_RGB', ETcVnColorSpaceTransform.TCVN_CST_BGR_TO_RGB);
AddLocalEnumeration('TCVN_CST_RGB_TO_BGR', ETcVnColorSpaceTransform.TCVN_CST_RGB_TO_BGR);
AddLocalEnumeration('TCVN_CST_BGRA_TO_RGBA', ETcVnColorSpaceTransform.TCVN_CST_BGRA_TO_RGBA);
AddLocalEnumeration('TCVN_CST_RGBA_TO_BGRA', ETcVnColorSpaceTransform.TCVN_CST_RGBA_TO_BGRA);
AddLocalEnumeration('TCVN_CST_BGR_TO_GRAY', ETcVnColorSpaceTransform.TCVN_CST_BGR_TO_GRAY);
AddLocalEnumeration('TCVN_CST_RGB_TO_GRAY', ETcVnColorSpaceTransform.TCVN_CST_RGB_TO_GRAY);
AddLocalEnumeration('TCVN_CST_GRAY_TO_BGR', ETcVnColorSpaceTransform.TCVN_CST_GRAY_TO_BGR);
AddLocalEnumeration('TCVN_CST_GRAY_TO_RGB', ETcVnColorSpaceTransform.TCVN_CST_GRAY_TO_RGB);
AddLocalEnumeration('TCVN_CST_GRAY_TO_BGRA', ETcVnColorSpaceTransform.TCVN_CST_GRAY_TO_BGRA);
AddLocalEnumeration('TCVN_CST_GRAY_TO_RGBA', ETcVnColorSpaceTransform.TCVN_CST_GRAY_TO_RGBA);
AddLocalEnumeration('TCVN_CST_BGRA_TO_GRAY', ETcVnColorSpaceTransform.TCVN_CST_BGRA_TO_GRAY);
AddLocalEnumeration('TCVN_CST_RGBA_TO_GRAY', ETcVnColorSpaceTransform.TCVN_CST_RGBA_TO_GRAY);
AddLocalEnumeration('TCVN_CST_RGB_TO_BGR_565', ETcVnColorSpaceTransform.TCVN_CST_RGB_TO_BGR_565);
AddLocalEnumeration('TCVN_CST_BGR_TO_BGR_565', ETcVnColorSpaceTransform.TCVN_CST_BGR_TO_BGR_565);
AddLocalEnumeration('TCVN_CST_BGR_565_TO_RGB', ETcVnColorSpaceTransform.TCVN_CST_BGR_565_TO_RGB);
AddLocalEnumeration('TCVN_CST_BGR_565_TO_BGR', ETcVnColorSpaceTransform.TCVN_CST_BGR_565_TO_BGR);
AddLocalEnumeration('TCVN_CST_RGBA_TO_BGR_565', ETcVnColorSpaceTransform.TCVN_CST_RGBA_TO_BGR_565);
AddLocalEnumeration('TCVN_CST_BGRA_TO_BGR_565', ETcVnColorSpaceTransform.TCVN_CST_BGRA_TO_BGR_565);
AddLocalEnumeration('TCVN_CST_BGR_565_TO_RGBA', ETcVnColorSpaceTransform.TCVN_CST_BGR_565_TO_RGBA);
AddLocalEnumeration('TCVN_CST_BGR_565_TO_BGRA', ETcVnColorSpaceTransform.TCVN_CST_BGR_565_TO_BGRA);
AddLocalEnumeration('TCVN_CST_GRAY_TO_BGR_565', ETcVnColorSpaceTransform.TCVN_CST_GRAY_TO_BGR_565);
AddLocalEnumeration('TCVN_CST_BGR_565_TO_GRAY', ETcVnColorSpaceTransform.TCVN_CST_BGR_565_TO_GRAY);
AddLocalEnumeration('TCVN_CST_RGB_TO_BGR_555', ETcVnColorSpaceTransform.TCVN_CST_RGB_TO_BGR_555);
AddLocalEnumeration('TCVN_CST_BGR_TO_BGR_555', ETcVnColorSpaceTransform.TCVN_CST_BGR_TO_BGR_555);
AddLocalEnumeration('TCVN_CST_BGR_555_TO_RGB', ETcVnColorSpaceTransform.TCVN_CST_BGR_555_TO_RGB);
AddLocalEnumeration('TCVN_CST_BGR_555_TO_BGR', ETcVnColorSpaceTransform.TCVN_CST_BGR_555_TO_BGR);
AddLocalEnumeration('TCVN_CST_RGBA_TO_BGR_555', ETcVnColorSpaceTransform.TCVN_CST_RGBA_TO_BGR_555);
AddLocalEnumeration('TCVN_CST_BGRA_TO_BGR_555', ETcVnColorSpaceTransform.TCVN_CST_BGRA_TO_BGR_555);
AddLocalEnumeration('TCVN_CST_BGR_555_TO_RGBA', ETcVnColorSpaceTransform.TCVN_CST_BGR_555_TO_RGBA);
AddLocalEnumeration('TCVN_CST_BGR_555_TO_BGRA', ETcVnColorSpaceTransform.TCVN_CST_BGR_555_TO_BGRA);
AddLocalEnumeration('TCVN_CST_GRAY_TO_BGR_555', ETcVnColorSpaceTransform.TCVN_CST_GRAY_TO_BGR_555);
AddLocalEnumeration('TCVN_CST_BGR_555_TO_GRAY', ETcVnColorSpaceTransform.TCVN_CST_BGR_555_TO_GRAY);
AddLocalEnumeration('TCVN_CST_BGR_TO_XYZ', ETcVnColorSpaceTransform.TCVN_CST_BGR_TO_XYZ);
AddLocalEnumeration('TCVN_CST_RGB_TO_XYZ', ETcVnColorSpaceTransform.TCVN_CST_RGB_TO_XYZ);
AddLocalEnumeration('TCVN_CST_XYZ_TO_BGR', ETcVnColorSpaceTransform.TCVN_CST_XYZ_TO_BGR);
AddLocalEnumeration('TCVN_CST_XYZ_TO_RGB', ETcVnColorSpaceTransform.TCVN_CST_XYZ_TO_RGB);
AddLocalEnumeration('TCVN_CST_BGR_TO_YCRCB', ETcVnColorSpaceTransform.TCVN_CST_BGR_TO_YCRCB);
AddLocalEnumeration('TCVN_CST_RGB_TO_YCRCB', ETcVnColorSpaceTransform.TCVN_CST_RGB_TO_YCRCB);
AddLocalEnumeration('TCVN_CST_YCRCB_TO_BGR', ETcVnColorSpaceTransform.TCVN_CST_YCRCB_TO_BGR);
AddLocalEnumeration('TCVN_CST_YCRCB_TO_RGB', ETcVnColorSpaceTransform.TCVN_CST_YCRCB_TO_RGB);
AddLocalEnumeration('TCVN_CST_BGR_TO_HSV', ETcVnColorSpaceTransform.TCVN_CST_BGR_TO_HSV);
AddLocalEnumeration('TCVN_CST_RGB_TO_HSV', ETcVnColorSpaceTransform.TCVN_CST_RGB_TO_HSV);
AddLocalEnumeration('TCVN_CST_BGR_TO_LAB', ETcVnColorSpaceTransform.TCVN_CST_BGR_TO_LAB);
AddLocalEnumeration('TCVN_CST_RGB_TO_LAB', ETcVnColorSpaceTransform.TCVN_CST_RGB_TO_LAB);
AddLocalEnumeration('TCVN_CST_BAYER_RG_TO_BGR', ETcVnColorSpaceTransform.TCVN_CST_BAYER_RG_TO_BGR);
AddLocalEnumeration('TCVN_CST_BAYER_BG_TO_RGB', ETcVnColorSpaceTransform.TCVN_CST_BAYER_BG_TO_RGB);
AddLocalEnumeration('TCVN_CST_BAYER_GR_TO_BGR', ETcVnColorSpaceTransform.TCVN_CST_BAYER_GR_TO_BGR);
AddLocalEnumeration('TCVN_CST_BAYER_GB_TO_RGB', ETcVnColorSpaceTransform.TCVN_CST_BAYER_GB_TO_RGB);
AddLocalEnumeration('TCVN_CST_BAYER_BG_TO_BGR', ETcVnColorSpaceTransform.TCVN_CST_BAYER_BG_TO_BGR);
AddLocalEnumeration('TCVN_CST_BAYER_RG_TO_RGB', ETcVnColorSpaceTransform.TCVN_CST_BAYER_RG_TO_RGB);
AddLocalEnumeration('TCVN_CST_BAYER_GB_TO_BGR', ETcVnColorSpaceTransform.TCVN_CST_BAYER_GB_TO_BGR);
AddLocalEnumeration('TCVN_CST_BAYER_GR_TO_RGB', ETcVnColorSpaceTransform.TCVN_CST_BAYER_GR_TO_RGB);
AddLocalEnumeration('TCVN_CST_BGR_TO_LUV', ETcVnColorSpaceTransform.TCVN_CST_BGR_TO_LUV);
AddLocalEnumeration('TCVN_CST_RGB_TO_LUV', ETcVnColorSpaceTransform.TCVN_CST_RGB_TO_LUV);
AddLocalEnumeration('TCVN_CST_BGR_TO_HLS', ETcVnColorSpaceTransform.TCVN_CST_BGR_TO_HLS);
AddLocalEnumeration('TCVN_CST_RGB_TO_HLS', ETcVnColorSpaceTransform.TCVN_CST_RGB_TO_HLS);
AddLocalEnumeration('TCVN_CST_HSV_TO_BGR', ETcVnColorSpaceTransform.TCVN_CST_HSV_TO_BGR);
AddLocalEnumeration('TCVN_CST_HSV_TO_RGB', ETcVnColorSpaceTransform.TCVN_CST_HSV_TO_RGB);
AddLocalEnumeration('TCVN_CST_LAB_TO_BGR', ETcVnColorSpaceTransform.TCVN_CST_LAB_TO_BGR);
AddLocalEnumeration('TCVN_CST_LAB_TO_RGB', ETcVnColorSpaceTransform.TCVN_CST_LAB_TO_RGB);
AddLocalEnumeration('TCVN_CST_LUV_TO_BGR', ETcVnColorSpaceTransform.TCVN_CST_LUV_TO_BGR);
AddLocalEnumeration('TCVN_CST_LUV_TO_RGB', ETcVnColorSpaceTransform.TCVN_CST_LUV_TO_RGB);
AddLocalEnumeration('TCVN_CST_HLS_TO_BGR', ETcVnColorSpaceTransform.TCVN_CST_HLS_TO_BGR);
AddLocalEnumeration('TCVN_CST_HLS_TO_RGB', ETcVnColorSpaceTransform.TCVN_CST_HLS_TO_RGB);
AddLocalEnumeration('TCVN_CST_BAYER_RG_TO_BGR_VNG', ETcVnColorSpaceTransform.TCVN_CST_BAYER_RG_TO_BGR_VNG);
AddLocalEnumeration('TCVN_CST_BAYER_GR_TO_BGR_VNG', ETcVnColorSpaceTransform.TCVN_CST_BAYER_GR_TO_BGR_VNG);
AddLocalEnumeration('TCVN_CST_BAYER_BG_TO_BGR_VNG', ETcVnColorSpaceTransform.TCVN_CST_BAYER_BG_TO_BGR_VNG);
AddLocalEnumeration('TCVN_CST_BAYER_GB_TO_BGR_VNG', ETcVnColorSpaceTransform.TCVN_CST_BAYER_GB_TO_BGR_VNG);
AddLocalEnumeration('TCVN_CST_BAYER_RG_TO_RGB_VNG', ETcVnColorSpaceTransform.TCVN_CST_BAYER_RG_TO_RGB_VNG);
AddLocalEnumeration('TCVN_CST_BAYER_GR_TO_RGB_VNG', ETcVnColorSpaceTransform.TCVN_CST_BAYER_GR_TO_RGB_VNG);
AddLocalEnumeration('TCVN_CST_BAYER_BG_TO_RGB_VNG', ETcVnColorSpaceTransform.TCVN_CST_BAYER_BG_TO_RGB_VNG);
AddLocalEnumeration('TCVN_CST_BAYER_GB_TO_RGB_VNG', ETcVnColorSpaceTransform.TCVN_CST_BAYER_GB_TO_RGB_VNG);
AddLocalEnumeration('TCVN_CST_BGR_TO_HSV_FULL', ETcVnColorSpaceTransform.TCVN_CST_BGR_TO_HSV_FULL);
AddLocalEnumeration('TCVN_CST_RGB_TO_HSV_FULL', ETcVnColorSpaceTransform.TCVN_CST_RGB_TO_HSV_FULL);
AddLocalEnumeration('TCVN_CST_BGR_TO_HLS_FULL', ETcVnColorSpaceTransform.TCVN_CST_BGR_TO_HLS_FULL);
AddLocalEnumeration('TCVN_CST_RGB_TO_HLS_FULL', ETcVnColorSpaceTransform.TCVN_CST_RGB_TO_HLS_FULL);
AddLocalEnumeration('TCVN_CST_HSV_TO_BGR_FULL', ETcVnColorSpaceTransform.TCVN_CST_HSV_TO_BGR_FULL);
AddLocalEnumeration('TCVN_CST_HSV_TO_RGB_FULL', ETcVnColorSpaceTransform.TCVN_CST_HSV_TO_RGB_FULL);
AddLocalEnumeration('TCVN_CST_HLS_TO_BGR_FULL', ETcVnColorSpaceTransform.TCVN_CST_HLS_TO_BGR_FULL);
AddLocalEnumeration('TCVN_CST_HLS_TO_RGB_FULL', ETcVnColorSpaceTransform.TCVN_CST_HLS_TO_RGB_FULL);
AddLocalEnumeration('TCVN_CST_LBGR_TO_LAB', ETcVnColorSpaceTransform.TCVN_CST_LBGR_TO_LAB);
AddLocalEnumeration('TCVN_CST_LRGB_TO_LAB', ETcVnColorSpaceTransform.TCVN_CST_LRGB_TO_LAB);
AddLocalEnumeration('TCVN_CST_LBGR_TO_LUV', ETcVnColorSpaceTransform.TCVN_CST_LBGR_TO_LUV);
AddLocalEnumeration('TCVN_CST_LRGB_TO_LUV', ETcVnColorSpaceTransform.TCVN_CST_LRGB_TO_LUV);
AddLocalEnumeration('TCVN_CST_LAB_TO_LBGR', ETcVnColorSpaceTransform.TCVN_CST_LAB_TO_LBGR);
AddLocalEnumeration('TCVN_CST_LAB_TO_LRGB', ETcVnColorSpaceTransform.TCVN_CST_LAB_TO_LRGB);
AddLocalEnumeration('TCVN_CST_LUV_TO_LBGR', ETcVnColorSpaceTransform.TCVN_CST_LUV_TO_LBGR);
AddLocalEnumeration('TCVN_CST_LUV_TO_LRGB', ETcVnColorSpaceTransform.TCVN_CST_LUV_TO_LRGB);
AddLocalEnumeration('TCVN_CST_BGR_TO_YUV', ETcVnColorSpaceTransform.TCVN_CST_BGR_TO_YUV);
AddLocalEnumeration('TCVN_CST_RGB_TO_YUV', ETcVnColorSpaceTransform.TCVN_CST_RGB_TO_YUV);
AddLocalEnumeration('TCVN_CST_YUV_TO_BGR', ETcVnColorSpaceTransform.TCVN_CST_YUV_TO_BGR);
AddLocalEnumeration('TCVN_CST_YUV_TO_RGB', ETcVnColorSpaceTransform.TCVN_CST_YUV_TO_RGB);
AddLocalEnumeration('TCVN_CST_BAYER_RG_TO_GRAY', ETcVnColorSpaceTransform.TCVN_CST_BAYER_RG_TO_GRAY);
AddLocalEnumeration('TCVN_CST_BAYER_GR_TO_GRAY', ETcVnColorSpaceTransform.TCVN_CST_BAYER_GR_TO_GRAY);
AddLocalEnumeration('TCVN_CST_BAYER_BG_TO_GRAY', ETcVnColorSpaceTransform.TCVN_CST_BAYER_BG_TO_GRAY);
AddLocalEnumeration('TCVN_CST_BAYER_GB_TO_GRAY', ETcVnColorSpaceTransform.TCVN_CST_BAYER_GB_TO_GRAY);
AddLocalEnumeration('TCVN_CST_YUV_420_NV12_TO_RGB', ETcVnColorSpaceTransform.TCVN_CST_YUV_420_NV12_TO_RGB);
AddLocalEnumeration('TCVN_CST_YUV_420_NV12_TO_BGR', ETcVnColorSpaceTransform.TCVN_CST_YUV_420_NV12_TO_BGR);
AddLocalEnumeration('TCVN_CST_YUV_420_NV21_TO_RGB', ETcVnColorSpaceTransform.TCVN_CST_YUV_420_NV21_TO_RGB);
AddLocalEnumeration('TCVN_CST_YUV_420_NV21_TO_BGR', ETcVnColorSpaceTransform.TCVN_CST_YUV_420_NV21_TO_BGR);
AddLocalEnumeration('TCVN_CST_YUV_420_SP_TO_RGB', ETcVnColorSpaceTransform.TCVN_CST_YUV_420_SP_TO_RGB);
AddLocalEnumeration('TCVN_CST_YUV_420_SP_TO_BGR', ETcVnColorSpaceTransform.TCVN_CST_YUV_420_SP_TO_BGR);
AddLocalEnumeration('TCVN_CST_YUV_420_NV12_TO_RGBA', ETcVnColorSpaceTransform.TCVN_CST_YUV_420_NV12_TO_RGBA);
AddLocalEnumeration('TCVN_CST_YUV_420_NV12_TO_BGRA', ETcVnColorSpaceTransform.TCVN_CST_YUV_420_NV12_TO_BGRA);
AddLocalEnumeration('TCVN_CST_YUV_420_NV21_TO_RGBA', ETcVnColorSpaceTransform.TCVN_CST_YUV_420_NV21_TO_RGBA);
AddLocalEnumeration('TCVN_CST_YUV_420_NV21_TO_BGRA', ETcVnColorSpaceTransform.TCVN_CST_YUV_420_NV21_TO_BGRA);
AddLocalEnumeration('TCVN_CST_YUV_420_SP_TO_RGBA', ETcVnColorSpaceTransform.TCVN_CST_YUV_420_SP_TO_RGBA);
AddLocalEnumeration('TCVN_CST_YUV_420_SP_TO_BGRA', ETcVnColorSpaceTransform.TCVN_CST_YUV_420_SP_TO_BGRA);
AddLocalEnumeration('TCVN_CST_YUV_420_YV12_TO_RGB', ETcVnColorSpaceTransform.TCVN_CST_YUV_420_YV12_TO_RGB);
AddLocalEnumeration('TCVN_CST_YUV_420_YV12_TO_BGR', ETcVnColorSpaceTransform.TCVN_CST_YUV_420_YV12_TO_BGR);
AddLocalEnumeration('TCVN_CST_YUV_420_IYUV_TO_RGB', ETcVnColorSpaceTransform.TCVN_CST_YUV_420_IYUV_TO_RGB);
AddLocalEnumeration('TCVN_CST_YUV_420_IYUV_TO_BGR', ETcVnColorSpaceTransform.TCVN_CST_YUV_420_IYUV_TO_BGR);
AddLocalEnumeration('TCVN_CST_YUV_420_I420_TO_RGB', ETcVnColorSpaceTransform.TCVN_CST_YUV_420_I420_TO_RGB);
AddLocalEnumeration('TCVN_CST_YUV_420_I420_TO_BGR', ETcVnColorSpaceTransform.TCVN_CST_YUV_420_I420_TO_BGR);
AddLocalEnumeration('TCVN_CST_YUV_420_P_TO_RGB', ETcVnColorSpaceTransform.TCVN_CST_YUV_420_P_TO_RGB);
AddLocalEnumeration('TCVN_CST_YUV_420_P_TO_BGR', ETcVnColorSpaceTransform.TCVN_CST_YUV_420_P_TO_BGR);
AddLocalEnumeration('TCVN_CST_YUV_420_YV12_TO_RGBA', ETcVnColorSpaceTransform.TCVN_CST_YUV_420_YV12_TO_RGBA);
AddLocalEnumeration('TCVN_CST_YUV_420_YV12_TO_BGRA', ETcVnColorSpaceTransform.TCVN_CST_YUV_420_YV12_TO_BGRA);
AddLocalEnumeration('TCVN_CST_YUV_420_IYUV_TO_RGBA', ETcVnColorSpaceTransform.TCVN_CST_YUV_420_IYUV_TO_RGBA);
AddLocalEnumeration('TCVN_CST_YUV_420_IYUV_TO_BGRA', ETcVnColorSpaceTransform.TCVN_CST_YUV_420_IYUV_TO_BGRA);
AddLocalEnumeration('TCVN_CST_YUV_420_I420_TO_RGBA', ETcVnColorSpaceTransform.TCVN_CST_YUV_420_I420_TO_RGBA);
AddLocalEnumeration('TCVN_CST_YUV_420_I420_TO_BGRA', ETcVnColorSpaceTransform.TCVN_CST_YUV_420_I420_TO_BGRA);
AddLocalEnumeration('TCVN_CST_YUV_420_P_TO_RGBA', ETcVnColorSpaceTransform.TCVN_CST_YUV_420_P_TO_RGBA);
AddLocalEnumeration('TCVN_CST_YUV_420_P_TO_BGRA', ETcVnColorSpaceTransform.TCVN_CST_YUV_420_P_TO_BGRA);
AddLocalEnumeration('TCVN_CST_YUV_420_TO_GRAY', ETcVnColorSpaceTransform.TCVN_CST_YUV_420_TO_GRAY);
AddLocalEnumeration('TCVN_CST_YUV_420_NV21_TO_GRAY', ETcVnColorSpaceTransform.TCVN_CST_YUV_420_NV21_TO_GRAY);
AddLocalEnumeration('TCVN_CST_YUV_420_NV12_TO_GRAY', ETcVnColorSpaceTransform.TCVN_CST_YUV_420_NV12_TO_GRAY);
AddLocalEnumeration('TCVN_CST_YUV_420_YV12_TO_GRAY', ETcVnColorSpaceTransform.TCVN_CST_YUV_420_YV12_TO_GRAY);
AddLocalEnumeration('TCVN_CST_YUV_420_IYUV_TO_GRAY', ETcVnColorSpaceTransform.TCVN_CST_YUV_420_IYUV_TO_GRAY);
AddLocalEnumeration('TCVN_CST_YUV_420_I420_TO_GRAY', ETcVnColorSpaceTransform.TCVN_CST_YUV_420_I420_TO_GRAY);
AddLocalEnumeration('TCVN_CST_YUV_420_SP_TO_GRAY', ETcVnColorSpaceTransform.TCVN_CST_YUV_420_SP_TO_GRAY);
AddLocalEnumeration('TCVN_CST_YUV_420_P_TO_GRAY', ETcVnColorSpaceTransform.TCVN_CST_YUV_420_P_TO_GRAY);
AddLocalEnumeration('TCVN_CST_YUV_422_UYVY_TO_RGB', ETcVnColorSpaceTransform.TCVN_CST_YUV_422_UYVY_TO_RGB);
AddLocalEnumeration('TCVN_CST_YUV_422_UYVY_TO_BGR', ETcVnColorSpaceTransform.TCVN_CST_YUV_422_UYVY_TO_BGR);
AddLocalEnumeration('TCVN_CST_YUV_422_Y422_TO_RGB', ETcVnColorSpaceTransform.TCVN_CST_YUV_422_Y422_TO_RGB);
AddLocalEnumeration('TCVN_CST_YUV_422_Y422_TO_BGR', ETcVnColorSpaceTransform.TCVN_CST_YUV_422_Y422_TO_BGR);
AddLocalEnumeration('TCVN_CST_YUV_422_UYNV_TO_RGB', ETcVnColorSpaceTransform.TCVN_CST_YUV_422_UYNV_TO_RGB);
AddLocalEnumeration('TCVN_CST_YUV_422_UYNV_TO_BGR', ETcVnColorSpaceTransform.TCVN_CST_YUV_422_UYNV_TO_BGR);
AddLocalEnumeration('TCVN_CST_YUV_422_UYVY_TO_RGBA', ETcVnColorSpaceTransform.TCVN_CST_YUV_422_UYVY_TO_RGBA);
AddLocalEnumeration('TCVN_CST_YUV_422_UYVY_TO_BGRA', ETcVnColorSpaceTransform.TCVN_CST_YUV_422_UYVY_TO_BGRA);
AddLocalEnumeration('TCVN_CST_YUV_422_Y422_TO_RGBA', ETcVnColorSpaceTransform.TCVN_CST_YUV_422_Y422_TO_RGBA);
AddLocalEnumeration('TCVN_CST_YUV_422_Y422_TO_BGRA', ETcVnColorSpaceTransform.TCVN_CST_YUV_422_Y422_TO_BGRA);
AddLocalEnumeration('TCVN_CST_YUV_422_UYNV_TO_RGBA', ETcVnColorSpaceTransform.TCVN_CST_YUV_422_UYNV_TO_RGBA);
AddLocalEnumeration('TCVN_CST_YUV_422_UYNV_TO_BGRA', ETcVnColorSpaceTransform.TCVN_CST_YUV_422_UYNV_TO_BGRA);
AddLocalEnumeration('TCVN_CST_YUV_422_YUY2_TO_RGB', ETcVnColorSpaceTransform.TCVN_CST_YUV_422_YUY2_TO_RGB);
AddLocalEnumeration('TCVN_CST_YUV_422_YUY2_TO_BGR', ETcVnColorSpaceTransform.TCVN_CST_YUV_422_YUY2_TO_BGR);
AddLocalEnumeration('TCVN_CST_YUV_422_YVYU_TO_RGB', ETcVnColorSpaceTransform.TCVN_CST_YUV_422_YVYU_TO_RGB);
AddLocalEnumeration('TCVN_CST_YUV_422_YVYU_TO_BGR', ETcVnColorSpaceTransform.TCVN_CST_YUV_422_YVYU_TO_BGR);
AddLocalEnumeration('TCVN_CST_YUV_422_YUYV_TO_RGB', ETcVnColorSpaceTransform.TCVN_CST_YUV_422_YUYV_TO_RGB);
AddLocalEnumeration('TCVN_CST_YUV_422_YUYV_TO_BGR', ETcVnColorSpaceTransform.TCVN_CST_YUV_422_YUYV_TO_BGR);
AddLocalEnumeration('TCVN_CST_YUV_422_YUNV_TO_RGB', ETcVnColorSpaceTransform.TCVN_CST_YUV_422_YUNV_TO_RGB);
AddLocalEnumeration('TCVN_CST_YUV_422_YUNV_TO_BGR', ETcVnColorSpaceTransform.TCVN_CST_YUV_422_YUNV_TO_BGR);
AddLocalEnumeration('TCVN_CST_YUV_422_YUY2_TO_RGBA', ETcVnColorSpaceTransform.TCVN_CST_YUV_422_YUY2_TO_RGBA);
AddLocalEnumeration('TCVN_CST_YUV_422_YUY2_TO_BGRA', ETcVnColorSpaceTransform.TCVN_CST_YUV_422_YUY2_TO_BGRA);
AddLocalEnumeration('TCVN_CST_YUV_422_YVYU_TO_RGBA', ETcVnColorSpaceTransform.TCVN_CST_YUV_422_YVYU_TO_RGBA);
AddLocalEnumeration('TCVN_CST_YUV_422_YVYU_TO_BGRA', ETcVnColorSpaceTransform.TCVN_CST_YUV_422_YVYU_TO_BGRA);
AddLocalEnumeration('TCVN_CST_YUV_422_YUYV_TO_RGBA', ETcVnColorSpaceTransform.TCVN_CST_YUV_422_YUYV_TO_RGBA);
AddLocalEnumeration('TCVN_CST_YUV_422_YUYV_TO_BGRA', ETcVnColorSpaceTransform.TCVN_CST_YUV_422_YUYV_TO_BGRA);
AddLocalEnumeration('TCVN_CST_YUV_422_YUNV_TO_RGBA', ETcVnColorSpaceTransform.TCVN_CST_YUV_422_YUNV_TO_RGBA);
AddLocalEnumeration('TCVN_CST_YUV_422_YUNV_TO_BGRA', ETcVnColorSpaceTransform.TCVN_CST_YUV_422_YUNV_TO_BGRA);
AddLocalEnumeration('TCVN_CST_YUV_422_UYVY_TO_GRAY', ETcVnColorSpaceTransform.TCVN_CST_YUV_422_UYVY_TO_GRAY);
AddLocalEnumeration('TCVN_CST_YUV_422_YUY2_TO_GRAY', ETcVnColorSpaceTransform.TCVN_CST_YUV_422_YUY2_TO_GRAY);
AddLocalEnumeration('TCVN_CST_YUV_422_Y422_TO_GRAY', ETcVnColorSpaceTransform.TCVN_CST_YUV_422_Y422_TO_GRAY);
AddLocalEnumeration('TCVN_CST_YUV_422_UYNV_TO_GRAY', ETcVnColorSpaceTransform.TCVN_CST_YUV_422_UYNV_TO_GRAY);
AddLocalEnumeration('TCVN_CST_YUV_422_YVYU_TO_GRAY', ETcVnColorSpaceTransform.TCVN_CST_YUV_422_YVYU_TO_GRAY);
AddLocalEnumeration('TCVN_CST_YUV_422_YUYV_TO_GRAY', ETcVnColorSpaceTransform.TCVN_CST_YUV_422_YUYV_TO_GRAY);
AddLocalEnumeration('TCVN_CST_YUV_422_YUNV_TO_GRAY', ETcVnColorSpaceTransform.TCVN_CST_YUV_422_YUNV_TO_GRAY);
AddLocalEnumeration('TCVN_CST_RGBA_TO_PREMULTIPLICATED_RGBA', ETcVnColorSpaceTransform.TCVN_CST_RGBA_TO_PREMULTIPLICATED_RGBA);
AddLocalEnumeration('TCVN_CST_PREMULTIPLICATED_RGBA_TO_RGBA', ETcVnColorSpaceTransform.TCVN_CST_PREMULTIPLICATED_RGBA_TO_RGBA);
AddLocalEnumeration('TCVN_CST_RGB_TO_YUV_420_I420', ETcVnColorSpaceTransform.TCVN_CST_RGB_TO_YUV_420_I420);
AddLocalEnumeration('TCVN_CST_BGR_TO_YUV_420_I420', ETcVnColorSpaceTransform.TCVN_CST_BGR_TO_YUV_420_I420);
AddLocalEnumeration('TCVN_CST_RGB_TO_YUV_420_IYUV', ETcVnColorSpaceTransform.TCVN_CST_RGB_TO_YUV_420_IYUV);
AddLocalEnumeration('TCVN_CST_BGR_TO_YUV_420_IYUV', ETcVnColorSpaceTransform.TCVN_CST_BGR_TO_YUV_420_IYUV);
AddLocalEnumeration('TCVN_CST_RGBA_TO_YUV_420_I420', ETcVnColorSpaceTransform.TCVN_CST_RGBA_TO_YUV_420_I420);
AddLocalEnumeration('TCVN_CST_BGRA_TO_YUV_420_I420', ETcVnColorSpaceTransform.TCVN_CST_BGRA_TO_YUV_420_I420);
AddLocalEnumeration('TCVN_CST_RGBA_TO_YUV_420_IYUV', ETcVnColorSpaceTransform.TCVN_CST_RGBA_TO_YUV_420_IYUV);
AddLocalEnumeration('TCVN_CST_BGRA_TO_YUV_420_IYUV', ETcVnColorSpaceTransform.TCVN_CST_BGRA_TO_YUV_420_IYUV);
AddLocalEnumeration('TCVN_CST_RGB_TO_YUV_420_YV12', ETcVnColorSpaceTransform.TCVN_CST_RGB_TO_YUV_420_YV12);
AddLocalEnumeration('TCVN_CST_BGR_TO_YUV_420_YV12', ETcVnColorSpaceTransform.TCVN_CST_BGR_TO_YUV_420_YV12);
AddLocalEnumeration('TCVN_CST_RGBA_TO_YUV_420_YV12', ETcVnColorSpaceTransform.TCVN_CST_RGBA_TO_YUV_420_YV12);
AddLocalEnumeration('TCVN_CST_BGRA_TO_YUV_420_YV12', ETcVnColorSpaceTransform.TCVN_CST_BGRA_TO_YUV_420_YV12);
AddLocalEnumeration('TCVN_CST_BAYER_RG_TO_BGR_EA', ETcVnColorSpaceTransform.TCVN_CST_BAYER_RG_TO_BGR_EA);
AddLocalEnumeration('TCVN_CST_BAYER_GR_TO_BGR_EA', ETcVnColorSpaceTransform.TCVN_CST_BAYER_GR_TO_BGR_EA);
AddLocalEnumeration('TCVN_CST_BAYER_BG_TO_BGR_EA', ETcVnColorSpaceTransform.TCVN_CST_BAYER_BG_TO_BGR_EA);
AddLocalEnumeration('TCVN_CST_BAYER_GB_TO_BGR_EA', ETcVnColorSpaceTransform.TCVN_CST_BAYER_GB_TO_BGR_EA);
AddLocalEnumeration('TCVN_CST_BAYER_RG_TO_RGB_EA', ETcVnColorSpaceTransform.TCVN_CST_BAYER_RG_TO_RGB_EA);
AddLocalEnumeration('TCVN_CST_BAYER_GR_TO_RGB_EA', ETcVnColorSpaceTransform.TCVN_CST_BAYER_GR_TO_RGB_EA);
AddLocalEnumeration('TCVN_CST_BAYER_BG_TO_RGB_EA', ETcVnColorSpaceTransform.TCVN_CST_BAYER_BG_TO_RGB_EA);
AddLocalEnumeration('TCVN_CST_BAYER_GB_TO_RGB_EA', ETcVnColorSpaceTransform.TCVN_CST_BAYER_GB_TO_RGB_EA);
AddLocalEnumeration('TCVN_CST_BAYER_RG_TO_BGRA', ETcVnColorSpaceTransform.TCVN_CST_BAYER_RG_TO_BGRA);
AddLocalEnumeration('TCVN_CST_BAYER_GR_TO_BGRA', ETcVnColorSpaceTransform.TCVN_CST_BAYER_GR_TO_BGRA);
AddLocalEnumeration('TCVN_CST_BAYER_BG_TO_BGRA', ETcVnColorSpaceTransform.TCVN_CST_BAYER_BG_TO_BGRA);
AddLocalEnumeration('TCVN_CST_BAYER_GB_TO_BGRA', ETcVnColorSpaceTransform.TCVN_CST_BAYER_GB_TO_BGRA);
AddLocalEnumeration('TCVN_CST_BAYER_RG_TO_RGBA', ETcVnColorSpaceTransform.TCVN_CST_BAYER_RG_TO_RGBA);
AddLocalEnumeration('TCVN_CST_BAYER_GR_TO_RGBA', ETcVnColorSpaceTransform.TCVN_CST_BAYER_GR_TO_RGBA);
AddLocalEnumeration('TCVN_CST_BAYER_BG_TO_RGBA', ETcVnColorSpaceTransform.TCVN_CST_BAYER_BG_TO_RGBA);
AddLocalEnumeration('TCVN_CST_BAYER_GB_TO_RGBA', ETcVnColorSpaceTransform.TCVN_CST_BAYER_GB_TO_RGBA);
AddLocalEnumeration('TCVN_CST_MAX', ETcVnColorSpaceTransform.TCVN_CST_MAX);
END_METHOD

METHOD PRIVATE AddLocalEnumeration
VAR_INPUT
	Enumeration : T_MAXSTRING;
	Value : ETcVnColorSpaceTransform;
END_VAR
AddEnumeration(Enumeration, Value);
END_METHOD

METHOD IsEnumeratorValueEqual : BOOL
VAR_INPUT
	Enumerator : I_KeyValueForwardEnumerator;
END_VAR
VAR
	storedValue : ETcVnColorSpaceTransform;
END_VAR
IF NOT Enumerator.TryGet(storedValue) THEN
	RETURN;
END_IF

IsEnumeratorValueEqual := storedValue = activeData;
END_METHOD

METHOD PUBLIC Clone : I_Datatype
VAR
    pClone : POINTER TO _ETcVnColorSpaceTransform;
END_VAR
pClone := __NEW(_ETcVnColorSpaceTransform(InitialValue := Value));
Clone := pClone^;
END_METHOD

PROPERTY PUBLIC Identifier : T_MAXSTRING
GET
Identifier := 'ETcVnColorSpaceTransform';
END_GET
END_PROPERTY

METHOD PUBLIC MakeReferenceTo
VAR_INPUT
	ReferenceTarget : REFERENCE TO ETcVnColorSpaceTransform;
END_VAR
activeData REF= ReferenceTarget;
SetBaseDatatypeReference();
END_METHOD

METHOD TryMakeReferenceTo : BOOL
VAR_INPUT
	Target : I_Datatype;
END_VAR
VAR
	targetAsEnum : I_EnumDatatype;
	pTargetData : POINTER TO ETcVnColorSpaceTransform;
END_VAR
IF NOT Target.TryResolveAsEnumDatatype(targetAsEnum) THEN
	RETURN;
END_IF

IF targetAsEnum.Identifier <> Identifier THEN
	RETURN;
END_IF

pTargetData := Target.Address;
activeData REF= pTargetData^;
SetBaseDatatypeReference();
TryMakeReferenceTo := TRUE;
END_METHOD

PROPERTY PUBLIC Value : ETcVnColorSpaceTransform
GET
Value := activeData;
END_GET
SET
activeData := Value;
END_SET
END_PROPERTY

END_FUNCTION_BLOCK

// Datatypes/Enums/_ETcVnColorTrainingMethod
{attribute 'linkalways'} 
{attribute 'no_explicit_call' := 'This FB is a CLASS and must be accessed using methods or properties'}
{attribute 'enable_dynamic_creation'}
FUNCTION_BLOCK _ETcVnColorTrainingMethod EXTENDS EnumDatatypeBase
VAR
	localData : ETcVnColorTrainingMethod;
	activeData : REFERENCE TO ETcVnColorTrainingMethod;
	enumBaseDatatype : _DINT(localData);
END_VAR

METHOD PROTECTED SetBaseDatatypeReference
VAR_INPUT
END_VAR
enumBaseDatatype.MakeReferenceTo(activeData);
END_METHOD

PROPERTY PUBLIC Address : PVOID
GET
Address := ADR(activeData);
END_GET
END_PROPERTY

METHOD PUBLIC ClearReference
VAR_INPUT
END_VAR
activeData REF= localData;
SetBaseDatatypeReference();
END_METHOD

PROPERTY PUBLIC Size : UDINT
GET
Size := SIZEOF(activeData);
END_GET
END_PROPERTY

METHOD FB_init : BOOL
VAR_INPUT
	bInitRetains : BOOL; // if TRUE, the retain variables are initialized (warm start / cold start)
	bInCopyCode : BOOL;  // if TRUE, the instance afterwards gets moved into the copy code (online change)
	InitialValue : ETcVnColorTrainingMethod;
END_VAR
localData := InitialValue;
AddBaseDatatype(enumBaseDatatype);
ClearReference();

AddLocalEnumeration('TCVN_CTM_LAB', ETcVnColorTrainingMethod.TCVN_CTM_LAB);
AddLocalEnumeration('TCVN_CTM_RGB', ETcVnColorTrainingMethod.TCVN_CTM_RGB);
END_METHOD

METHOD PRIVATE AddLocalEnumeration
VAR_INPUT
	Enumeration : T_MAXSTRING;
	Value : ETcVnColorTrainingMethod;
END_VAR
AddEnumeration(Enumeration, Value);
END_METHOD

METHOD IsEnumeratorValueEqual : BOOL
VAR_INPUT
	Enumerator : I_KeyValueForwardEnumerator;
END_VAR
VAR
	storedValue : ETcVnColorTrainingMethod;
END_VAR
IF NOT Enumerator.TryGet(storedValue) THEN
	RETURN;
END_IF

